C03640=1088.865,407.445,399.289,177.788,26.148,154.195
C03641=1088.871,407.692,399.248,177.791,26.157,154.197
C03642=1088.878,407.938,399.208,177.795,26.166,154.199
C03643=1088.884,408.185,399.168,177.797,26.175,154.200
C03644=1088.890,408.432,399.127,177.800,26.183,154.202
C03645=1088.896,408.678,399.087,177.804,26.192,154.204
C03646=1088.903,408.925,399.047,177.807,26.201,154.206
C03647=1088.909,409.172,399.006,177.811,26.210,154.207
C03648=1088.915,409.419,398.966,177.815,26.219,154.209
C03649=1088.922,409.665,398.925,177.818,26.227,154.211
C03650=1088.927,409.911,398.884,177.821,26.236,154.213
C03651=1088.934,410.158,398.844,177.824,26.245,154.215
C03652=1088.940,410.404,398.804,177.828,26.254,154.217
C03653=1088.946,410.652,398.763,177.831,26.263,154.218
C03654=1088.953,410.879,398.726,177.834,26.272,154.220
C03655=1088.958,411.106,398.688,177.837,26.280,154.222
C03656=1088.963,411.333,398.651,177.841,26.288,154.223
C03657=1088.969,411.560,398.613,177.844,26.297,154.225
C03658=1088.976,411.787,398.575,177.847,26.305,154.227
C03659=1088.981,412.014,398.538,177.850,26.313,154.228
C03660=1088.987,412.241,398.500,177.852,26.322,154.230
C03661=1088.993,412.469,398.463,177.855,26.330,154.232
C03662=1089.000,412.716,398.422,177.859,26.339,154.234
C03663=1089.006,412.962,398.381,177.863,26.349,154.236
C03664=1089.012,413.209,398.340,177.866,26.358,154.238
C03665=1089.019,413.455,398.299,177.869,26.368,154.240
C03666=1089.025,413.702,398.258,177.873,26.377,154.241
C03667=1089.032,413.948,398.218,177.876,26.386,154.243
C03668=1089.038,414.195,398.176,177.880,26.395,154.245
C03669=1089.045,414.441,398.136,177.883,26.405,154.247
C03670=1089.051,414.688,398.094,177.886,26.414,154.249
C03671=1089.058,414.934,398.053,177.890,26.423,154.251
C03672=1089.063,415.181,398.012,177.894,26.433,154.253
C03673=1089.071,415.428,397.971,177.896,26.442,154.255
C03674=1089.077,415.674,397.930,177.900,26.452,154.257
C03675=1089.084,415.921,397.889,177.904,26.462,154.259
C03676=1089.090,416.167,397.848,177.908,26.471,154.261
C03677=1089.096,416.413,397.806,177.910,26.481,154.263
C03678=1089.103,416.660,397.765,177.914,26.490,154.265
C03679=1089.109,416.906,397.723,177.918,26.500,154.267
C03680=1089.115,417.153,397.682,177.921,26.510,154.269
C03681=1089.122,417.399,397.641,177.924,26.520,154.271
C03682=1089.128,417.645,397.599,177.928,26.529,154.273
C03683=1089.135,417.892,397.557,177.931,26.539,154.275
C03684=1089.140,418.138,397.516,177.935,26.549,154.277
C03685=1089.148,418.385,397.475,177.939,26.559,154.279
C03686=1089.154,418.631,397.433,177.941,26.569,154.281
C03687=1089.160,418.878,397.391,177.945,26.579,154.283
C03688=1089.166,419.124,397.350,177.949,26.589,154.285
C03689=1089.173,419.371,397.308,177.952,26.599,154.288
C03690=1089.179,419.617,397.267,177.956,26.609,154.290
C03691=1089.186,419.864,397.226,177.960,26.619,154.292
C03692=1089.192,420.110,397.183,177.963,26.630,154.294
C03693=1089.199,420.356,397.142,177.966,26.639,154.296
C03694=1089.205,420.603,397.100,177.970,26.649,154.298
C03695=1089.211,420.850,397.058,177.973,26.660,154.300
C03696=1089.219,421.096,397.016,177.977,26.670,154.302
C03697=1089.225,421.342,396.975,177.980,26.680,154.305
C03698=1089.231,421.589,396.933,177.984,26.691,154.307
C03699=1089.238,421.834,396.891,177.988,26.701,154.309
C03700=1089.244,422.081,396.849,177.991,26.711,154.311
C03701=1089.251,422.327,396.806,177.995,26.722,154.313
C03702=1089.257,422.574,396.765,177.998,26.732,154.316
C03703=1089.264,422.820,396.722,178.002,26.743,154.318
C03704=1089.270,423.067,396.681,178.006,26.753,154.320
C03705=1089.277,423.312,396.638,178.009,26.764,154.322
C03706=1089.283,423.559,396.597,178.013,26.775,154.324
C03707=1089.290,423.806,396.554,178.016,26.785,154.327
C03708=1089.296,424.051,396.512,178.020,26.796,154.329
C03709=1089.303,424.298,396.470,178.023,26.807,154.331
C03710=1089.311,424.618,396.415,178.027,26.820,154.334
C03711=1089.319,424.939,396.360,178.032,26.834,154.337
C03712=1089.328,425.259,396.305,178.037,26.849,154.340
C03713=1089.336,425.580,396.250,178.042,26.863,154.343
C03714=1089.343,425.825,396.207,178.045,26.874,154.346
C03715=1089.349,426.071,396.165,178.049,26.884,154.348
C03716=1089.356,426.318,396.122,178.052,26.895,154.350
C03717=1089.363,426.564,396.080,178.056,26.906,154.353
C03718=1089.369,426.811,396.037,178.059,26.918,154.355
C03719=1089.376,427.056,395.994,178.063,26.928,154.357
C03720=1089.382,427.302,395.952,178.067,26.940,154.360
C03721=1089.389,427.549,395.909,178.071,26.951,154.362
C03722=1089.396,427.795,395.867,178.074,26.962,154.365
C03723=1089.402,428.042,395.824,178.078,26.973,154.367
C03724=1089.409,428.288,395.781,178.081,26.985,154.369
C03725=1089.415,428.533,395.739,178.085,26.996,154.372
C03726=1089.422,428.780,395.696,178.088,27.007,154.374
C03727=1089.429,429.026,395.653,178.093,27.019,154.377
C03728=1089.436,429.272,395.610,178.096,27.030,154.379
C03729=1089.442,429.518,395.568,178.100,27.041,154.382
C03730=1089.448,429.765,395.524,178.103,27.053,154.384
C03731=1089.456,430.011,395.481,178.107,27.065,154.387
C03732=1089.462,430.257,395.438,178.111,27.076,154.389
C03733=1089.469,430.503,395.395,178.115,27.088,154.392
C03734=1089.474,430.749,395.352,178.118,27.099,154.394
C03735=1089.481,430.995,395.309,178.121,27.111,154.397
C03736=1089.488,431.241,395.266,178.125,27.123,154.399
C03737=1089.495,431.487,395.223,178.129,27.135,154.402
C03738=1089.502,431.733,395.180,178.133,27.146,154.404
C03739=1089.508,431.979,395.137,178.136,27.158,154.407
C03740=1089.515,432.225,395.093,178.141,27.171,154.410
C03741=1089.521,432.472,395.050,178.144,27.182,154.412
C03742=1089.528,432.717,395.007,178.147,27.194,154.415
C03743=1089.535,432.963,394.963,178.151,27.206,154.418
C03744=1089.542,433.210,394.921,178.155,27.218,154.420
C03745=1089.548,433.456,394.877,178.159,27.231,154.423
C03746=1089.554,433.702,394.833,178.162,27.242,154.426
C03747=1089.562,433.947,394.790,178.166,27.255,154.428
C03748=1089.568,434.194,394.747,178.170,27.267,154.431
C03749=1089.575,434.441,394.702,178.173,27.279,154.434
C03750=1089.586,434.835,394.632,178.180,27.300,154.438
C03751=1089.596,435.230,394.562,178.186,27.319,154.442
C03752=1089.607,435.626,394.492,178.192,27.339,154.447
C03753=1089.617,436.021,394.422,178.198,27.359,154.451
C03754=1089.624,436.266,394.378,178.202,27.372,154.454
C03755=1089.631,436.512,394.334,178.205,27.385,154.457
C03756=1089.638,436.759,394.290,178.209,27.398,154.460
C03757=1089.645,437.004,394.246,178.213,27.410,154.463
C03758=1089.651,437.250,394.202,178.217,27.423,154.465
C03759=1089.658,437.496,394.159,178.220,27.436,154.468
C03760=1089.664,437.742,394.114,178.225,27.449,154.471
C03761=1089.671,437.988,394.070,178.228,27.461,154.474
C03762=1089.680,438.310,394.013,178.234,27.479,154.478
C03763=1089.689,438.630,393.955,178.238,27.495,154.481
C03764=1089.698,438.952,393.897,178.244,27.512,154.485
C03765=1089.707,439.273,393.839,178.248,27.529,154.489
C03766=1089.714,439.519,393.796,178.252,27.543,154.492
C03767=1089.720,439.764,393.751,178.256,27.556,154.495
C03768=1089.728,440.010,393.707,178.260,27.569,154.498
C03769=1089.735,440.256,393.663,178.264,27.583,154.501
C03770=1089.742,440.501,393.618,178.268,27.596,154.504
C03771=1089.748,440.748,393.574,178.272,27.609,154.507
C03772=1089.755,440.993,393.529,178.275,27.623,154.510
C03773=1089.762,441.240,393.485,178.279,27.637,154.513
C03774=1089.768,441.485,393.440,178.284,27.650,154.516
C03775=1089.775,441.731,393.396,178.287,27.664,154.519
C03776=1089.782,441.977,393.351,178.291,27.677,154.522
C03777=1089.789,442.222,393.306,178.296,27.691,154.525
C03778=1089.797,442.468,393.261,178.299,27.705,154.529
C03779=1089.803,442.714,393.217,178.303,27.719,154.532
C03780=1089.810,442.959,393.173,178.307,27.733,154.535
C03781=1089.816,443.206,393.127,178.311,27.747,154.538
C03782=1089.823,443.451,393.083,178.315,27.761,154.541
C03783=1089.830,443.697,393.038,178.319,27.775,154.544
C03784=1089.837,443.943,392.993,178.323,27.789,154.547
C03785=1089.844,444.189,392.948,178.327,27.803,154.551
C03786=1089.851,444.434,392.902,178.331,27.817,154.554
C03787=1089.858,444.680,392.857,178.335,27.832,154.557
C03788=1089.865,444.925,392.813,178.338,27.846,154.560
C03789=1089.872,445.171,392.768,178.342,27.860,154.564
C03790=1089.879,445.418,392.722,178.345,27.874,154.567
C03791=1089.886,445.662,392.677,178.348,27.888,154.570
C03792=1089.893,445.908,392.632,178.351,27.903,154.574
C03793=1089.899,446.154,392.587,178.354,27.917,154.577
C03794=1089.907,446.399,392.541,178.356,27.931,154.580
C03795=1089.913,446.646,392.496,178.358,27.945,154.584
C03796=1089.920,446.891,392.451,178.361,27.959,154.587
C03797=1089.928,447.137,392.406,178.363,27.973,154.591
C03798=1089.934,447.383,392.360,178.364,27.987,154.594
C03799=1089.941,447.628,392.315,178.366,28.001,154.597
C03800=1089.948,447.874,392.269,178.367,28.015,154.601
C03801=1089.956,448.119,392.224,178.368,28.030,154.604
C03802=1089.962,448.366,392.178,178.370,28.043,154.608
C03803=1089.969,448.611,392.133,178.371,28.058,154.611
C03804=1089.976,448.857,392.087,178.372,28.071,154.615
C03805=1089.983,449.102,392.042,178.373,28.086,154.618
C03806=1089.990,449.347,391.996,178.373,28.100,154.622
C03807=1089.997,449.593,391.950,178.374,28.114,154.625
C03808=1090.004,449.838,391.906,178.374,28.128,154.629
C03809=1090.015,450.084,391.861,178.374,28.140,154.632
C03810=1089.633,450.077,391.673,178.332,28.336,154.686
C03811=1089.623,449.830,391.716,178.331,28.323,154.682
C03812=1089.615,449.585,391.762,178.330,28.310,154.679
C03813=1089.609,449.340,391.808,178.330,28.295,154.675
C03814=1089.602,449.095,391.853,178.329,28.281,154.672
C03815=1089.594,448.849,391.898,178.329,28.267,154.669
C03816=1089.587,448.603,391.944,178.327,28.253,154.665
C03817=1089.580,448.358,391.990,178.326,28.239,154.662
C03818=1089.573,448.111,392.036,178.325,28.225,154.658
C03819=1089.566,447.867,392.081,178.324,28.211,154.655
C03820=1089.559,447.620,392.126,178.322,28.197,154.651
C03821=1089.552,447.375,392.172,178.320,28.183,154.648
C03822=1089.545,447.128,392.218,178.318,28.169,154.644
C03823=1089.538,446.884,392.263,178.316,28.154,154.641
C03824=1089.532,446.637,392.308,178.314,28.140,154.637
C03825=1089.524,446.392,392.354,178.311,28.126,154.634
C03826=1089.517,446.146,392.399,178.309,28.111,154.631
C03827=1089.510,445.901,392.445,178.306,28.097,154.627
C03828=1089.503,445.655,392.490,178.303,28.083,154.624
C03829=1089.497,445.409,392.535,178.300,28.069,154.621
C03830=1089.489,445.164,392.581,178.296,28.055,154.617
C03831=1089.482,444.918,392.626,178.293,28.040,154.614
C03832=1089.475,444.672,392.670,178.289,28.027,154.611
C03833=1089.468,444.426,392.716,178.285,28.012,154.607
C03834=1089.462,444.181,392.761,178.281,27.998,154.604
C03835=1089.454,443.935,392.806,178.277,27.984,154.601
C03836=1089.448,443.690,392.850,178.273,27.969,154.598
C03837=1089.441,443.443,392.896,178.269,27.955,154.595
C03838=1089.434,443.198,392.940,178.264,27.941,154.591
C03839=1089.427,442.952,392.985,178.261,27.927,154.588
C03840=1089.420,442.707,393.030,178.257,27.913,154.585
C03841=1089.413,442.460,393.075,178.252,27.899,154.582
C03842=1089.406,442.215,393.119,178.249,27.886,154.579
C03843=1089.400,441.969,393.165,178.245,27.872,154.576
C03844=1089.393,441.723,393.210,178.240,27.858,154.573
C03845=1089.385,441.477,393.255,178.237,27.844,154.570
C03846=1089.379,441.232,393.299,178.233,27.831,154.567
C03847=1089.372,440.986,393.343,178.229,27.817,154.563
C03848=1089.365,440.740,393.388,178.225,27.803,154.560
C03849=1089.358,440.495,393.432,178.220,27.790,154.557
C03850=1089.351,440.249,393.477,178.217,27.777,154.554
C03851=1089.345,440.003,393.521,178.213,27.763,154.551
C03852=1089.338,439.757,393.566,178.209,27.750,154.548
C03853=1089.331,439.511,393.610,178.205,27.736,154.545
C03854=1089.324,439.265,393.655,178.201,27.723,154.542
C03855=1089.315,438.957,393.710,178.196,27.707,154.539
C03856=1089.307,438.648,393.765,178.191,27.690,154.535
C03857=1089.298,438.340,393.821,178.186,27.674,154.531
C03858=1089.290,438.031,393.876,178.181,27.658,154.528
C03859=1089.283,437.785,393.920,178.177,27.645,154.525
C03860=1089.275,437.540,393.964,178.174,27.632,154.522
C03861=1089.269,437.294,394.008,178.169,27.619,154.519
C03862=1089.262,437.048,394.052,178.166,27.606,154.516
C03863=1089.255,436.801,394.096,178.162,27.593,154.514
C03864=1089.249,436.556,394.141,178.158,27.581,154.511
C03865=1089.241,436.310,394.184,178.154,27.568,154.508
C03866=1089.235,436.064,394.228,178.150,27.555,154.505
C03867=1089.229,435.818,394.272,178.146,27.543,154.502
C03868=1089.222,435.572,394.316,178.142,27.530,154.500
C03869=1089.214,435.326,394.359,178.139,27.518,154.497
C03870=1089.208,435.080,394.403,178.135,27.505,154.494
C03871=1089.202,434.834,394.447,178.131,27.493,154.491
C03872=1089.195,434.588,394.491,178.127,27.480,154.489
C03873=1089.188,434.342,394.534,178.124,27.468,154.486
C03874=1089.181,434.096,394.578,178.119,27.456,154.483
C03875=1089.175,433.850,394.622,178.116,27.443,154.480
C03876=1089.168,433.605,394.665,178.112,27.431,154.478
C03877=1089.161,433.359,394.709,178.108,27.419,154.475
C03878=1089.155,433.112,394.752,178.104,27.407,154.472
C03879=1089.149,432.866,394.796,178.101,27.394,154.470
C03880=1089.141,432.620,394.840,178.096,27.382,154.467
C03881=1089.135,432.373,394.883,178.093,27.371,154.464
C03882=1089.128,432.127,394.926,178.089,27.358,154.462
C03883=1089.121,431.882,394.970,178.085,27.346,154.459
C03884=1089.115,431.635,395.012,178.081,27.335,154.457
C03885=1089.108,431.389,395.056,178.078,27.323,154.454
C03886=1089.101,431.143,395.099,178.074,27.311,154.451
C03887=1089.094,430.897,395.142,178.071,27.299,154.449
C03888=1089.088,430.651,395.185,178.066,27.287,154.446
C03889=1089.081,430.405,395.228,178.063,27.276,154.444
C03890=1089.075,430.158,395.271,178.059,27.264,154.441
C03891=1089.068,429.913,395.315,178.056,27.253,154.439
C03892=1089.062,429.667,395.357,178.051,27.241,154.436
C03893=1089.055,429.421,395.400,178.048,27.230,154.434
C03894=1089.048,429.175,395.443,178.044,27.218,154.431
C03895=1089.042,428.928,395.486,178.041,27.206,154.429
C03896=1089.035,428.682,395.529,178.037,27.195,154.426
C03897=1089.028,428.436,395.572,178.033,27.184,154.424
C03898=1089.022,428.190,395.615,178.030,27.172,154.421
C03899=1089.015,427.944,395.658,178.025,27.161,154.419
C03900=1089.008,427.697,395.700,178.022,27.150,154.417
C03901=1089.001,427.451,395.743,178.018,27.139,154.414
C03902=1088.996,427.205,395.786,178.015,27.128,154.412
C03903=1088.989,426.959,395.828,178.011,27.116,154.409
C03904=1088.982,426.713,395.871,178.007,27.106,154.407
C03905=1088.975,426.466,395.913,178.004,27.094,154.405
C03906=1088.968,426.220,395.956,178.000,27.083,154.402
C03907=1088.962,425.984,395.996,177.996,27.073,154.400
C03908=1088.956,425.750,396.037,177.993,27.062,154.398
C03909=1088.950,425.514,396.078,177.989,27.052,154.396
C03910=1088.944,425.279,396.118,177.986,27.042,154.393
C03911=1088.937,425.044,396.159,177.983,27.031,154.391
C03912=1088.931,424.809,396.199,177.979,27.021,154.389
C03913=1088.925,424.572,396.240,177.975,27.010,154.387
C03914=1088.919,424.337,396.281,177.972,27.000,154.384
C03915=1088.912,424.091,396.323,177.969,26.989,154.382
C03916=1088.906,423.845,396.365,177.965,26.979,154.380
C03917=1088.899,423.598,396.407,177.962,26.968,154.378
C03918=1088.893,423.353,396.449,177.958,26.958,154.375
C03919=1088.886,423.106,396.492,177.954,26.947,154.373
C03920=1088.879,422.859,396.534,177.951,26.936,154.371
C03921=1088.873,422.614,396.576,177.947,26.925,154.369
C03922=1088.867,422.367,396.618,177.943,26.915,154.366
C03923=1088.860,422.121,396.660,177.940,26.904,154.364
C03924=1088.854,421.874,396.702,177.936,26.894,154.362
C03925=1088.847,421.628,396.744,177.932,26.884,154.360
C03926=1088.840,421.381,396.786,177.929,26.873,154.358
C03927=1088.834,421.136,396.828,177.925,26.863,154.355
C03928=1088.828,420.889,396.870,177.921,26.853,154.353
C03929=1088.821,420.643,396.911,177.918,26.843,154.351
C03930=1088.814,420.397,396.953,177.915,26.832,154.349
C03931=1088.807,420.150,396.995,177.911,26.822,154.347
C03932=1088.802,419.903,397.037,177.907,26.812,154.345
C03933=1088.795,419.657,397.079,177.904,26.802,154.343
C03934=1088.789,419.411,397.121,177.900,26.792,154.341
C03935=1088.781,419.164,397.162,177.896,26.781,154.338
C03936=1088.775,418.918,397.203,177.894,26.772,154.336
C03937=1088.769,418.671,397.245,177.890,26.762,154.334
C03938=1088.763,418.425,397.287,177.886,26.752,154.332
C03939=1088.756,418.178,397.328,177.882,26.742,154.330
C03940=1088.750,417.932,397.369,177.879,26.732,154.328
C03941=1088.743,417.685,397.411,177.876,26.722,154.326
C03942=1088.737,417.439,397.453,177.872,26.712,154.324
C03943=1088.730,417.181,397.497,177.869,26.702,154.322
C03944=1088.723,416.924,397.539,177.865,26.691,154.320
C03945=1088.717,416.666,397.583,177.861,26.681,154.317
C03946=1088.710,416.408,397.627,177.858,26.671,154.315
C03947=1088.704,416.162,397.668,177.854,26.661,154.313
C03948=1088.698,415.915,397.708,177.850,26.652,154.311
C03949=1088.691,415.669,397.750,177.847,26.643,154.309
C03950=1088.684,415.423,397.791,177.844,26.633,154.307
C03951=1088.678,415.176,397.833,177.840,26.623,154.305
C03952=1088.671,414.930,397.874,177.837,26.614,154.303
C03953=1088.665,414.682,397.915,177.833,26.604,154.301
C03954=1088.658,414.436,397.956,177.829,26.595,154.300
C03955=1088.652,414.190,397.998,177.826,26.585,154.298
C03956=1088.645,413.943,398.038,177.823,26.576,154.296
C03957=1088.639,413.697,398.079,177.819,26.567,154.294
C03958=1088.632,413.450,398.120,177.816,26.557,154.292
C03959=1088.626,413.204,398.161,177.812,26.548,154.290
C03960=1088.620,412.957,398.202,177.809,26.539,154.288
C03961=1088.613,412.710,398.243,177.806,26.530,154.286
C03962=1088.607,412.464,398.284,177.802,26.520,154.284
C03963=1088.602,412.241,398.320,177.799,26.512,154.283
C03964=1088.595,412.020,398.357,177.796,26.504,154.281
C03965=1088.589,411.798,398.394,177.793,26.495,154.279
C03966=1088.584,411.575,398.430,177.790,26.487,154.278
C03967=1088.578,411.353,398.467,177.787,26.479,154.276
C03968=1088.572,411.131,398.504,177.784,26.471,154.274
C03969=1088.567,410.909,398.540,177.780,26.463,154.273
C03970=1088.561,410.687,398.578,177.777,26.455,154.271
C03971=1088.555,410.440,398.618,177.774,26.445,154.269
C03972=1088.548,410.194,398.659,177.771,26.437,154.267
C03973=1088.542,409.948,398.699,177.767,26.427,154.265
C03974=1088.535,409.700,398.740,177.764,26.419,154.264
C03975=1088.529,409.454,398.780,177.760,26.410,154.262
C03976=1088.523,409.207,398.821,177.757,26.401,154.260
C03977=1088.517,408.961,398.862,177.753,26.392,154.258
C03978=1088.510,408.715,398.902,177.750,26.383,154.256
C03979=1088.505,408.468,398.943,177.747,26.374,154.255
C03980=1088.498,408.221,398.983,177.744,26.365,154.253
C03981=1088.492,407.975,399.023,177.740,26.357,154.251
C03982=1088.486,407.727,399.064,177.737,26.348,154.249
C03983=1088.479,407.481,399.104,177.733,26.339,154.247
C03984=1088.473,407.234,399.144,177.730,26.331,154.246
C03985=1088.467,406.988,399.184,177.726,26.321,154.244
C03986=1088.460,406.741,399.225,177.723,26.313,154.242
C03987=1088.455,406.494,399.265,177.720,26.305,154.241
C03988=1088.448,406.248,399.305,177.716,26.296,154.239
C03989=1088.442,406.001,399.346,177.713,26.288,154.237
C03990=1088.435,405.755,399.386,177.710,26.278,154.235
C03991=1088.429,405.508,399.425,177.707,26.271,154.234
C03992=1088.423,405.261,399.465,177.704,26.262,154.232
C03993=1088.416,405.014,399.506,177.700,26.254,154.230
C03994=1088.410,404.767,399.546,177.697,26.245,154.229
C03995=1088.403,404.520,399.585,177.693,26.236,154.227
C03996=1088.397,404.274,399.626,177.690,26.228,154.225
C03997=1088.391,404.027,399.666,177.687,26.220,154.224
C03998=1088.384,403.781,399.706,177.683,26.211,154.222
C03999=1088.378,403.534,399.745,177.680,26.203,154.220
C04000=1088.372,403.287,399.785,177.677,26.195,154.219
C04001=1088.366,403.040,399.825,177.673,26.187,154.217
C04002=1088.359,402.794,399.865,177.670,26.178,154.215
C04003=1088.353,402.547,399.905,177.667,26.171,154.214
C04004=1088.347,402.300,399.945,177.663,26.162,154.212
C04005=1088.341,402.054,399.984,177.660,26.154,154.211
C04006=1088.335,401.807,400.024,177.657,26.146,154.209
C04007=1088.329,401.560,400.064,177.653,26.138,154.207
C04008=1088.322,401.314,400.103,177.650,26.130,154.206
C04009=1088.316,401.066,400.142,177.647,26.122,154.204
C04010=1088.309,400.820,400.182,177.644,26.114,154.203
C04011=1088.303,400.573,400.222,177.640,26.106,154.201
C04012=1088.297,400.326,400.262,177.637,26.098,154.200
C04013=1088.291,400.079,400.301,177.634,26.090,154.198
C04014=1088.285,399.833,400.340,177.631,26.082,154.196
C04015=1088.278,399.587,400.380,177.627,26.074,154.195
C04016=1088.272,399.339,400.419,177.624,26.066,154.193
C04017=1088.266,399.092,400.459,177.621,26.058,154.192
C04018=1088.260,398.845,400.498,177.618,26.050,154.190
C04019=1088.255,398.618,400.534,177.615,26.043,154.189
C04020=1088.249,398.392,400.571,177.611,26.036,154.187
C04021=1088.243,398.164,400.607,177.608,26.029,154.186
C04022=1088.237,397.938,400.643,177.606,26.022,154.185
C04023=1088.231,397.711,400.679,177.603,26.015,154.183
C04024=1088.225,397.483,400.715,177.600,26.007,154.182
C04025=1088.220,397.256,400.751,177.596,26.000,154.181
C04026=1088.214,397.029,400.787,177.593,25.993,154.179
C04027=1088.208,396.782,400.826,177.590,25.985,154.178
C04028=1088.202,396.535,400.866,177.587,25.978,154.176
C04029=1088.195,396.288,400.904,177.584,25.970,154.175
C04030=1088.190,396.041,400.944,177.581,25.963,154.173
C04031=1088.183,395.795,400.982,177.578,25.955,154.172
C04032=1088.177,395.547,401.022,177.574,25.947,154.170
C04033=1088.171,395.301,401.061,177.570,25.940,154.169
C04034=1088.164,395.054,401.100,177.567,25.932,154.167
C04035=1088.158,394.807,401.139,177.564,25.925,154.166
C04036=1088.152,394.561,401.178,177.561,25.917,154.165
C04037=1088.146,394.314,401.217,177.558,25.910,154.163
C04038=1088.139,394.067,401.256,177.555,25.902,154.162
C04039=1088.134,393.820,401.294,177.552,25.895,154.160
C04040=1088.127,393.573,401.333,177.548,25.888,154.159
C04041=1088.121,393.326,401.372,177.545,25.880,154.157
C04042=1088.115,393.080,401.411,177.541,25.873,154.156
C04043=1088.109,392.832,401.449,177.538,25.866,154.155
C04044=1088.103,392.586,401.488,177.535,25.858,154.153
C04045=1088.096,392.339,401.527,177.532,25.851,154.152
C04046=1088.091,392.092,401.565,177.529,25.844,154.150
C04047=1088.084,391.845,401.604,177.526,25.836,154.149
C04048=1088.077,391.598,401.643,177.522,25.829,154.148
C04049=1088.072,391.352,401.681,177.519,25.822,154.146
C04050=1088.065,391.105,401.720,177.516,25.815,154.145
C04051=1088.060,390.858,401.758,177.512,25.807,154.144
C04052=1088.053,390.611,401.797,177.509,25.800,154.142
C04053=1088.046,390.364,401.836,177.506,25.793,154.141
C04054=1088.041,390.117,401.874,177.502,25.786,154.140
C04055=1088.034,389.870,401.913,177.499,25.779,154.138
C04056=1088.028,389.624,401.951,177.496,25.772,154.137
C04057=1088.022,389.376,401.989,177.493,25.765,154.136
C04058=1088.015,389.130,402.027,177.490,25.758,154.134
C04059=1088.009,388.883,402.065,177.486,25.751,154.133
C04060=1088.003,388.636,402.104,177.483,25.744,154.132
C04061=1087.997,388.389,402.142,177.480,25.737,154.131
C04062=1087.991,388.142,402.180,177.477,25.730,154.129
C04063=1087.985,387.896,402.219,177.474,25.723,154.128
C04064=1087.978,387.648,402.257,177.470,25.716,154.127
C04065=1087.972,387.402,402.295,177.467,25.709,154.125
C04066=1087.966,387.155,402.333,177.464,25.703,154.124
C04067=1087.960,386.908,402.372,177.461,25.696,154.123
C04068=1087.954,386.661,402.410,177.458,25.689,154.122
C04069=1087.948,386.414,402.448,177.454,25.682,154.120
C04070=1087.942,386.167,402.485,177.451,25.675,154.119
C04071=1087.936,385.921,402.524,177.448,25.668,154.118
C04072=1087.929,385.673,402.562,177.445,25.661,154.116
C04073=1087.923,385.427,402.600,177.441,25.655,154.115
C04074=1087.918,385.180,402.638,177.438,25.648,154.114
C04075=1087.912,384.959,402.672,177.435,25.641,154.113
C04076=1087.907,384.738,402.706,177.432,25.636,154.112
C04077=1087.901,384.519,402.739,177.430,25.630,154.111
C04078=1087.896,384.297,402.773,177.426,25.623,154.110
C04079=1087.891,384.077,402.807,177.424,25.618,154.108
C04080=1087.886,383.857,402.841,177.421,25.611,154.107
C04081=1087.879,383.637,402.874,177.418,25.606,154.106
C04082=1087.874,383.417,402.909,177.416,25.600,154.105
C04083=1087.868,383.170,402.946,177.412,25.593,154.104
C04084=1087.862,382.922,402.984,177.409,25.586,154.103
C04085=1087.856,382.675,403.022,177.406,25.580,154.102
C04086=1087.850,382.429,403.059,177.403,25.573,154.100
C04087=1087.844,382.181,403.097,177.399,25.566,154.099
C04088=1087.838,381.934,403.135,177.396,25.560,154.098
C04089=1087.831,381.688,403.172,177.393,25.554,154.097
C04090=1087.826,381.441,403.210,177.389,25.547,154.096
C04091=1087.819,381.193,403.247,177.386,25.540,154.095
C04092=1087.813,380.946,403.285,177.383,25.534,154.093
C04093=1087.807,380.700,403.322,177.380,25.528,154.092
C04094=1087.801,380.453,403.359,177.377,25.521,154.091
C04095=1087.795,380.205,403.398,177.374,25.515,154.090
C04096=1087.789,379.958,403.435,177.370,25.509,154.089
C04097=1087.783,379.711,403.472,177.367,25.502,154.088
C04098=1087.777,379.465,403.510,177.364,25.496,154.087
C04099=1087.771,379.218,403.547,177.360,25.489,154.085
C04100=1087.764,378.970,403.585,177.357,25.483,154.084
C04101=1087.758,378.723,403.622,177.355,25.477,154.083
C04102=1087.752,378.476,403.659,177.351,25.471,154.082
C04103=1087.746,378.229,403.697,177.348,25.464,154.081
C04104=1087.741,377.982,403.734,177.345,25.458,154.080
C04105=1087.734,377.735,403.771,177.342,25.451,154.079
C04106=1087.728,377.487,403.808,177.338,25.445,154.077
C04107=1087.722,377.241,403.846,177.335,25.439,154.076
C04108=1087.716,376.994,403.882,177.332,25.433,154.075
C04109=1087.710,376.747,403.920,177.329,25.427,154.074
C04110=1087.704,376.500,403.957,177.326,25.420,154.073
C04111=1087.698,376.252,403.994,177.322,25.414,154.072
C04112=1087.692,376.006,404.031,177.319,25.408,154.071
C04113=1087.686,375.758,404.068,177.317,25.402,154.070
C04114=1087.680,375.511,404.105,177.313,25.396,154.069
C04115=1087.674,375.265,404.143,177.310,25.389,154.068
C04116=1087.668,375.017,404.180,177.306,25.383,154.067
C04117=1087.662,374.770,404.216,177.303,25.377,154.066
C04118=1087.656,374.523,404.253,177.301,25.371,154.064
C04119=1087.651,374.276,404.291,177.297,25.365,154.063
C04120=1087.644,374.029,404.327,177.294,25.358,154.062
C04121=1087.638,373.781,404.365,177.291,25.353,154.061
C04122=1087.632,373.534,404.401,177.287,25.347,154.060
C04123=1087.625,373.287,404.438,177.285,25.341,154.059
C04124=1087.620,373.039,404.475,177.281,25.335,154.058
C04125=1087.613,372.792,404.511,177.278,25.329,154.057
C04126=1087.608,372.546,404.549,177.275,25.323,154.056
C04127=1087.601,372.299,404.585,177.272,25.317,154.055
C04128=1087.595,372.052,404.622,177.269,25.311,154.054
C04129=1087.589,371.804,404.659,177.265,25.305,154.053
C04130=1087.583,371.557,404.695,177.262,25.299,154.052
C04131=1087.573,371.144,404.756,177.257,25.289,154.050
C04132=1087.563,370.731,404.818,177.251,25.279,154.049
C04133=1087.553,370.318,404.879,177.247,25.270,154.047
C04134=1087.543,369.906,404.940,177.241,25.260,154.045
C04135=1087.536,369.659,404.976,177.238,25.254,154.044
C04136=1087.531,369.411,405.012,177.234,25.248,154.043
C04137=1087.525,369.164,405.049,177.231,25.242,154.042
C04138=1087.518,368.917,405.085,177.229,25.237,154.041
C04139=1087.513,368.669,405.122,177.225,25.231,154.040
C04140=1087.507,368.422,405.158,177.222,25.225,154.039
C04141=1087.501,368.175,405.194,177.219,25.220,154.038
C04142=1087.495,367.928,405.231,177.216,25.214,154.037
C04143=1087.489,367.681,405.268,177.212,25.208,154.036
C04144=1087.483,367.433,405.303,177.210,25.202,154.035
C04145=1087.477,367.186,405.340,177.206,25.197,154.034
C04146=1087.471,366.939,405.377,177.203,25.191,154.034
C04147=1087.466,366.692,405.412,177.200,25.186,154.033
C04148=1087.459,366.445,405.449,177.197,25.179,154.032
C04149=1087.453,366.197,405.484,177.194,25.174,154.031
C04150=1087.448,365.950,405.521,177.191,25.168,154.030
C04151=1087.442,365.702,405.557,177.188,25.163,154.029
C04152=1087.436,365.456,405.593,177.184,25.157,154.028
C04153=1087.430,365.208,405.629,177.182,25.151,154.027
C04154=1087.424,364.961,405.665,177.178,25.146,154.026
C04155=1087.418,364.713,405.701,177.175,25.140,154.025
C04156=1087.411,364.466,405.738,177.172,25.135,154.024
C04157=1087.405,364.219,405.773,177.169,25.129,154.023
C04158=1087.400,363.972,405.810,177.165,25.124,154.022
C04159=1087.394,363.724,405.846,177.163,25.118,154.021
C04160=1087.388,363.477,405.881,177.159,25.113,154.020
C04161=1087.382,363.229,405.918,177.156,25.107,154.020
C04162=1087.376,362.982,405.954,177.153,25.102,154.019
C04163=1087.370,362.735,405.989,177.150,25.096,154.018
C04164=1087.364,362.488,406.025,177.146,25.091,154.017
C04165=1087.358,362.240,406.061,177.143,25.086,154.016
C04166=1087.352,361.992,406.097,177.140,25.080,154.015
C04167=1087.347,361.745,406.132,177.137,25.075,154.014
C04168=1087.339,361.499,406.168,177.134,25.069,154.013
C04169=1087.333,361.251,406.204,177.130,25.064,154.013
C04170=1087.327,361.003,406.240,177.128,25.059,154.012
C04171=1087.322,360.756,406.275,177.124,25.053,154.011
C04172=1087.316,360.509,406.311,177.122,25.048,154.010
C04173=1087.310,360.262,406.347,177.118,25.042,154.009
C04174=1087.304,360.015,406.382,177.115,25.037,154.008
C04175=1087.298,359.767,406.418,177.112,25.032,154.007
C04176=1087.292,359.519,406.454,177.109,25.026,154.006
C04177=1087.287,359.272,406.489,177.106,25.021,154.006
C04178=1087.280,359.025,406.524,177.102,25.016,154.005
C04179=1087.274,358.777,406.560,177.099,25.010,154.004
C04180=1087.268,358.530,406.596,177.096,25.005,154.003
C04181=1087.262,358.283,406.631,177.093,25.000,154.002
C04182=1087.256,358.035,406.667,177.090,24.995,154.001
C04183=1087.247,357.638,406.723,177.084,24.986,154.000
C04184=1087.237,357.241,406.780,177.080,24.978,153.999
C04185=1087.227,356.843,406.837,177.075,24.970,153.997
C04186=1087.218,356.446,406.894,177.069,24.961,153.996
C04187=1087.212,356.199,406.929,177.067,24.956,153.995
C04188=1087.206,355.952,406.965,177.063,24.951,153.994
C04189=1087.200,355.705,406.999,177.061,24.946,153.993
C04190=1087.195,355.457,407.034,177.057,24.941,153.993
C04191=1087.189,355.209,407.070,177.054,24.936,153.992
C04192=1087.182,354.962,407.105,177.051,24.930,153.991
C04193=1087.176,354.715,407.141,177.048,24.926,153.990
C04194=1087.171,354.467,407.175,177.045,24.920,153.989
C04195=1087.164,354.220,407.210,177.042,24.915,153.989
C04196=1087.159,353.973,407.246,177.038,24.910,153.988
C04197=1087.153,353.724,407.281,177.036,24.905,153.987
C04198=1087.147,353.478,407.316,177.032,24.900,153.986
C04199=1087.141,353.230,407.351,177.030,24.895,153.985
C04200=1087.136,352.982,407.386,177.026,24.890,153.985
C04201=1087.129,352.735,407.421,177.023,24.885,153.984
C04202=1087.124,352.487,407.456,177.020,24.880,153.983
C04203=1087.117,352.240,407.491,177.017,24.875,153.982
C04204=1087.112,351.992,407.526,177.013,24.870,153.982
C04205=1087.105,351.745,407.561,177.011,24.865,153.981
C04206=1087.100,351.498,407.595,177.007,24.860,153.980
C04207=1087.094,351.250,407.630,177.005,24.855,153.979
C04208=1087.088,351.003,407.665,177.001,24.850,153.979
C04209=1087.082,350.755,407.700,176.998,24.845,153.978
C04210=1087.077,350.508,407.735,176.995,24.840,153.977
C04211=1087.070,350.260,407.769,176.992,24.836,153.976
C04212=1087.065,350.013,407.805,176.988,24.830,153.975
C04213=1087.058,349.765,407.839,176.986,24.826,153.975
C04214=1087.053,349.518,407.874,176.982,24.820,153.974
C04215=1087.046,349.270,407.909,176.979,24.816,153.973
C04216=1087.040,349.022,407.943,176.976,24.811,153.972
C04217=1087.035,348.775,407.978,176.973,24.806,153.972
C04218=1087.029,348.527,408.013,176.970,24.801,153.971
C04219=1087.023,348.280,408.047,176.967,24.796,153.970
C04220=1087.017,348.032,408.082,176.964,24.792,153.969
C04221=1087.011,347.785,408.116,176.961,24.786,153.969
C04222=1087.006,347.538,408.151,176.958,24.782,153.968
C04223=1086.999,347.290,408.186,176.954,24.777,153.967
C04224=1086.993,347.042,408.220,176.951,24.772,153.967
C04225=1086.988,346.794,408.255,176.948,24.767,153.966
C04226=1086.982,346.547,408.289,176.945,24.762,153.965
C04227=1086.976,346.300,408.323,176.942,24.758,153.964
C04228=1086.970,346.051,408.358,176.939,24.753,153.964
C04229=1086.964,345.805,408.393,176.936,24.748,153.963
C04230=1086.958,345.557,408.427,176.932,24.743,153.962
C04231=1086.952,345.309,408.462,176.930,24.739,153.962
C04232=1086.947,345.062,408.496,176.927,24.734,153.961
C04233=1086.941,344.814,408.530,176.923,24.729,153.960
C04234=1086.934,344.566,408.564,176.921,24.724,153.959
C04235=1086.925,344.172,408.618,176.916,24.717,153.958
C04236=1086.916,343.778,408.673,176.911,24.710,153.957
C04237=1086.906,343.383,408.728,176.906,24.702,153.956
C04238=1086.897,342.989,408.782,176.901,24.695,153.955
C04239=1086.891,342.741,408.816,176.897,24.690,153.954
C04240=1086.885,342.494,408.850,176.895,24.685,153.954
C04241=1086.880,342.246,408.885,176.892,24.681,153.953
C04242=1086.874,341.999,408.919,176.888,24.676,153.952
C04243=1086.868,341.751,408.952,176.885,24.672,153.952
C04244=1086.862,341.503,408.987,176.883,24.667,153.951
C04245=1086.856,341.255,409.021,176.879,24.662,153.950
C04246=1086.850,341.008,409.055,176.876,24.658,153.950
C04247=1086.844,340.760,409.088,176.873,24.653,153.949
C04248=1086.839,340.513,409.122,176.870,24.648,153.948
C04249=1086.832,340.265,409.156,176.867,24.644,153.948
C04250=1086.827,340.017,409.190,176.863,24.640,153.947
C04251=1086.821,339.770,409.224,176.861,24.635,153.946
C04252=1086.815,339.522,409.258,176.858,24.631,153.946
C04253=1086.809,339.275,409.291,176.854,24.626,153.945
C04254=1086.803,339.027,409.326,176.851,24.621,153.944
C04255=1086.797,338.779,409.360,176.849,24.617,153.944
C04256=1086.791,338.531,409.393,176.845,24.612,153.943
C04257=1086.786,338.284,409.427,176.842,24.608,153.942
C04258=1086.780,338.036,409.460,176.839,24.604,153.942
C04259=1086.774,337.789,409.495,176.836,24.599,153.941
C04260=1086.768,337.540,409.528,176.833,24.594,153.940
C04261=1086.762,337.293,409.562,176.830,24.590,153.940
C04262=1086.757,337.045,409.596,176.827,24.585,153.939
C04263=1086.751,336.798,409.630,176.824,24.581,153.938
C04264=1086.745,336.550,409.663,176.821,24.577,153.938
C04265=1086.739,336.303,409.696,176.818,24.572,153.937
C04266=1086.733,336.055,409.730,176.814,24.568,153.937
C04267=1086.727,335.807,409.763,176.812,24.564,153.936
C04268=1086.721,335.559,409.798,176.809,24.559,153.935
C04269=1086.715,335.311,409.831,176.805,24.555,153.935
C04270=1086.709,335.064,409.864,176.802,24.550,153.934
C04271=1086.703,334.816,409.898,176.799,24.546,153.933
C04272=1086.698,334.568,409.931,176.796,24.541,153.933
C04273=1086.692,334.321,409.964,176.793,24.537,153.932
C04274=1086.686,334.073,409.998,176.790,24.533,153.932
C04275=1086.680,333.826,410.031,176.788,24.528,153.931
C04276=1086.674,333.578,410.064,176.784,24.524,153.930
C04277=1086.669,333.330,410.098,176.781,24.519,153.930
C04278=1086.663,333.083,410.132,176.778,24.515,153.929
C04279=1086.657,332.835,410.165,176.775,24.511,153.928
C04280=1086.651,332.587,410.198,176.772,24.507,153.928
C04281=1086.646,332.339,410.231,176.769,24.502,153.927
C04282=1086.640,332.091,410.265,176.766,24.498,153.927
C04283=1086.634,331.844,410.297,176.763,24.494,153.926
C04284=1086.628,331.596,410.331,176.760,24.489,153.925
C04285=1086.622,331.348,410.365,176.757,24.485,153.925
C04286=1086.616,331.101,410.398,176.754,24.481,153.924
C04287=1086.606,330.700,410.451,176.749,24.475,153.923
C04288=1086.596,330.300,410.504,176.744,24.467,153.922
C04289=1086.587,329.900,410.558,176.739,24.461,153.922
C04290=1086.577,329.500,410.611,176.733,24.454,153.921
C04291=1086.571,329.252,410.644,176.731,24.450,153.920
C04292=1086.566,329.004,410.677,176.728,24.446,153.920
C04293=1086.559,328.757,410.710,176.725,24.442,153.919
C04294=1086.554,328.509,410.743,176.722,24.438,153.918
C04295=1086.547,328.261,410.776,176.718,24.433,153.918
C04296=1086.541,328.013,410.808,176.715,24.429,153.917
C04297=1086.536,327.765,410.841,176.713,24.425,153.917
C04298=1086.530,327.518,410.874,176.710,24.421,153.916
C04299=1086.524,327.270,410.907,176.706,24.417,153.916
C04300=1086.518,327.022,410.940,176.703,24.412,153.915
C04301=1086.511,326.774,410.973,176.700,24.408,153.914
C04302=1086.507,326.527,411.005,176.698,24.404,153.914
C04303=1086.501,326.279,411.038,176.695,24.400,153.913
C04304=1086.495,326.031,411.071,176.692,24.396,153.913
C04305=1086.489,325.784,411.104,176.688,24.392,153.912
C04306=1086.483,325.535,411.136,176.685,24.388,153.912
C04307=1086.477,325.287,411.169,176.682,24.384,153.911
C04308=1086.471,325.040,411.202,176.679,24.380,153.911
C04309=1086.465,324.792,411.234,176.677,24.376,153.910
C04310=1086.460,324.544,411.267,176.673,24.371,153.910
C04311=1086.454,324.297,411.300,176.670,24.367,153.909
C04312=1086.448,324.049,411.332,176.667,24.363,153.908
C04313=1086.442,323.801,411.365,176.664,24.359,153.908
C04314=1086.436,323.552,411.397,176.661,24.355,153.907
C04315=1086.430,323.305,411.430,176.659,24.351,153.907
C04316=1086.425,323.058,411.463,176.655,24.347,153.906
C04317=1086.419,322.809,411.495,176.652,24.343,153.906
C04318=1086.413,322.562,411.528,176.649,24.339,153.905
C04319=1086.407,322.313,411.560,176.646,24.335,153.905
C04320=1086.402,322.066,411.593,176.643,24.331,153.904
C04321=1086.396,321.818,411.625,176.640,24.327,153.904
C04322=1086.389,321.571,411.657,176.638,24.323,153.903
C04323=1086.384,321.322,411.690,176.634,24.319,153.903
C04324=1086.379,321.075,411.722,176.631,24.314,153.902
C04325=1086.372,320.827,411.754,176.628,24.310,153.901
C04326=1086.367,320.578,411.787,176.625,24.306,153.901
C04327=1086.361,320.332,411.819,176.622,24.303,153.901
C04328=1086.355,320.083,411.852,176.619,24.299,153.900
C04329=1086.349,319.835,411.884,176.617,24.295,153.899
C04330=1086.343,319.588,411.916,176.614,24.291,153.899
C04331=1086.339,319.340,411.949,176.610,24.286,153.898
C04332=1086.333,319.092,411.981,176.607,24.282,153.898
C04333=1086.327,318.845,412.013,176.604,24.279,153.897
C04334=1086.321,318.596,412.045,176.601,24.275,153.897
C04335=1086.316,318.348,412.078,176.598,24.271,153.896
C04336=1086.310,318.100,412.109,176.596,24.267,153.896
C04337=1086.304,317.853,412.142,176.593,24.263,153.895
C04338=1086.298,317.605,412.174,176.590,24.259,153.895
C04339=1086.289,317.198,412.226,176.585,24.252,153.894
C04340=1086.280,316.790,412.279,176.580,24.246,153.893
C04341=1086.270,316.384,412.332,176.574,24.239,153.892
C04342=1086.261,315.977,412.385,176.570,24.233,153.891
C04343=1086.256,315.729,412.417,176.567,24.229,153.891
C04344=1086.250,315.481,412.449,176.564,24.225,153.890
C04345=1086.244,315.234,412.480,176.561,24.221,153.890
C04346=1086.238,314.986,412.512,176.558,24.217,153.889
C04347=1086.233,314.738,412.544,176.555,24.213,153.889
C04348=1086.227,314.490,412.576,176.552,24.209,153.888
C04349=1086.221,314.242,412.608,176.549,24.205,153.888
C04350=1086.215,313.994,412.640,176.546,24.202,153.887
C04351=1086.209,313.746,412.671,176.543,24.198,153.887
C04352=1086.203,313.498,412.703,176.540,24.194,153.886
C04353=1086.197,313.250,412.735,176.537,24.190,153.886
C04354=1086.191,313.002,412.767,176.534,24.187,153.886
C04355=1086.185,312.755,412.798,176.531,24.183,153.885
C04356=1086.179,312.507,412.830,176.529,24.179,153.885
C04357=1086.174,312.258,412.861,176.526,24.176,153.884
C04358=1086.168,312.010,412.893,176.523,24.172,153.884
C04359=1086.161,311.763,412.924,176.519,24.167,153.883
C04360=1086.156,311.515,412.956,176.516,24.164,153.883
C04361=1086.150,311.267,412.988,176.513,24.160,153.882
C04362=1086.144,311.020,413.019,176.510,24.156,153.882
C04363=1086.138,310.771,413.050,176.507,24.153,153.881
C04364=1086.133,310.523,413.082,176.504,24.149,153.881
C04365=1086.127,310.275,413.114,176.501,24.145,153.880
C04366=1086.121,310.028,413.145,176.498,24.142,153.880
C04367=1086.115,309.780,413.177,176.495,24.138,153.880
C04368=1086.110,309.532,413.208,176.492,24.134,153.879
C04369=1086.103,309.284,413.240,176.489,24.130,153.879
C04370=1086.098,309.036,413.271,176.486,24.127,153.878
C04371=1086.092,308.787,413.303,176.484,24.123,153.878
C04372=1086.086,308.540,413.334,176.481,24.119,153.877
C04373=1086.080,308.292,413.366,176.478,24.116,153.877
C04374=1086.074,308.044,413.396,176.475,24.112,153.876
C04375=1086.068,307.796,413.428,176.472,24.108,153.876
C04376=1086.063,307.548,413.460,176.469,24.104,153.875
C04377=1086.057,307.300,413.490,176.466,24.101,153.875
C04378=1086.051,307.052,413.522,176.463,24.097,153.875
C04379=1086.046,306.804,413.553,176.460,24.093,153.874
C04380=1086.040,306.557,413.584,176.457,24.090,153.874
C04381=1086.034,306.308,413.615,176.454,24.086,153.873
C04382=1086.028,306.061,413.646,176.451,24.083,153.873
C04383=1086.022,305.812,413.678,176.448,24.078,153.872
C04384=1086.016,305.565,413.709,176.445,24.075,153.872
C04385=1086.011,305.317,413.740,176.442,24.071,153.872
C04386=1086.005,305.069,413.772,176.439,24.067,153.871
C04387=1085.999,304.821,413.802,176.436,24.063,153.871
C04388=1085.994,304.573,413.834,176.433,24.060,153.870
C04389=1085.988,304.325,413.864,176.430,24.056,153.870
C04390=1085.982,304.077,413.896,176.427,24.053,153.869
C04391=1085.973,303.673,413.946,176.422,24.047,153.869
C04392=1085.963,303.269,413.996,176.417,24.040,153.868
C04393=1085.954,302.865,414.047,176.413,24.035,153.867
C04394=1085.945,302.461,414.097,176.408,24.028,153.866
C04395=1085.939,302.213,414.129,176.405,24.025,153.866
C04396=1085.934,301.965,414.160,176.402,24.021,153.866
C04397=1085.928,301.717,414.190,176.399,24.018,153.865
C04398=1085.923,301.469,414.221,176.396,24.014,153.865
C04399=1085.916,301.221,414.252,176.393,24.010,153.864
C04400=1085.911,300.973,414.283,176.391,24.007,153.864
C04401=1085.905,300.725,414.314,176.388,24.003,153.863
C04402=1085.900,300.477,414.345,176.385,24.000,153.863
C04403=1085.894,300.229,414.375,176.382,23.996,153.862
C04404=1085.889,299.982,414.407,176.379,23.992,153.862
C04405=1085.882,299.733,414.437,176.376,23.989,153.862
C04406=1085.877,299.485,414.468,176.373,23.985,153.861
C04407=1085.872,299.237,414.499,176.370,23.981,153.861
C04408=1085.866,298.989,414.529,176.367,23.978,153.860
C04409=1085.861,298.741,414.560,176.364,23.974,153.860
C04410=1085.855,298.493,414.590,176.362,23.970,153.859
C04411=1085.850,298.245,414.621,176.359,23.967,153.859
C04412=1085.843,297.997,414.652,176.356,23.963,153.859
C04413=1085.837,297.749,414.682,176.353,23.960,153.858
C04414=1085.832,297.501,414.713,176.350,23.956,153.858
C04415=1085.827,297.253,414.744,176.347,23.953,153.857
C04416=1085.821,297.005,414.774,176.344,23.949,153.857
C04417=1085.815,296.757,414.804,176.341,23.945,153.857
C04418=1085.809,296.509,414.835,176.338,23.942,153.856
C04419=1085.803,296.261,414.866,176.335,23.938,153.856
C04420=1085.798,296.013,414.896,176.332,23.935,153.855
C04421=1085.792,295.765,414.927,176.330,23.931,153.855
C04422=1085.786,295.517,414.957,176.327,23.928,153.854
C04423=1085.780,295.269,414.987,176.324,23.924,153.854
C04424=1085.775,295.021,415.017,176.321,23.921,153.854
C04425=1085.768,294.772,415.048,176.318,23.918,153.853
C04426=1085.763,294.524,415.079,176.315,23.914,153.853
C04427=1085.757,294.276,415.109,176.312,23.910,153.853
C04428=1085.752,294.028,415.139,176.309,23.907,153.852
C04429=1085.746,293.780,415.169,176.306,23.903,153.852
C04430=1085.740,293.532,415.199,176.303,23.900,153.851
C04431=1085.734,293.285,415.230,176.300,23.896,153.851
C04432=1085.729,293.036,415.259,176.297,23.893,153.851
C04433=1085.723,292.788,415.290,176.295,23.890,153.850
C04434=1085.717,292.540,415.320,176.292,23.886,153.850
C04435=1085.711,292.293,415.351,176.289,23.882,153.849
C04436=1085.706,292.044,415.380,176.286,23.879,153.849
C04437=1085.699,291.796,415.411,176.283,23.876,153.849
C04438=1085.694,291.548,415.441,176.280,23.872,153.848
C04439=1085.688,291.299,415.471,176.277,23.869,153.848
C04440=1085.682,291.052,415.501,176.274,23.865,153.847
C04441=1085.677,290.803,415.531,176.271,23.861,153.847
C04442=1085.671,290.555,415.561,176.269,23.859,153.847
C04443=1085.662,290.165,415.609,176.264,23.853,153.846
C04444=1085.653,289.776,415.656,176.259,23.847,153.846
C04445=1085.645,289.386,415.702,176.255,23.842,153.845
C04446=1085.635,288.995,415.750,176.250,23.837,153.844
C04447=1085.629,288.747,415.780,176.247,23.833,153.844
C04448=1085.624,288.499,415.810,176.244,23.830,153.844
C04449=1085.618,288.251,415.839,176.242,23.827,153.843
C04450=1085.612,288.003,415.869,176.239,23.823,153.843
C04451=1085.606,287.755,415.899,176.236,23.820,153.843
C04452=1085.600,287.507,415.929,176.233,23.816,153.842
C04453=1085.595,287.258,415.959,176.230,23.813,153.842
C04454=1085.589,287.010,415.988,176.227,23.810,153.841
C04455=1085.583,286.762,416.018,176.224,23.806,153.841
C04456=1085.578,286.515,416.047,176.222,23.803,153.841
C04457=1085.572,286.266,416.077,176.219,23.800,153.840
C04458=1085.566,286.018,416.107,176.216,23.796,153.840
C04459=1085.560,285.770,416.136,176.213,23.793,153.839
C04460=1085.555,285.522,416.166,176.210,23.789,153.839
C04461=1085.549,285.274,416.196,176.207,23.786,153.839
C04462=1085.543,285.026,416.226,176.204,23.782,153.838
C04463=1085.537,284.777,416.255,176.202,23.780,153.838
C04464=1085.532,284.529,416.285,176.199,23.776,153.838
C04465=1085.526,284.281,416.314,176.196,23.772,153.837
C04466=1085.520,284.033,416.345,176.193,23.769,153.837
C04467=1085.514,283.785,416.374,176.190,23.766,153.837
C04468=1085.509,283.537,416.403,176.187,23.762,153.836
C04469=1085.504,283.288,416.432,176.185,23.759,153.836
C04470=1085.498,283.040,416.462,176.182,23.756,153.835
C04471=1085.492,282.792,416.491,176.179,23.753,153.835
C04472=1085.486,282.543,416.521,176.176,23.749,153.835
C04473=1085.481,282.296,416.551,176.173,23.745,153.834
C04474=1085.475,282.048,416.580,176.170,23.742,153.834
C04475=1085.469,281.800,416.609,176.168,23.739,153.834
C04476=1085.464,281.551,416.639,176.165,23.735,153.833
C04477=1085.458,281.303,416.668,176.162,23.732,153.833
C04478=1085.452,281.055,416.698,176.159,23.729,153.833
C04479=1085.447,280.806,416.727,176.156,23.726,153.832
C04480=1085.441,280.559,416.756,176.154,23.722,153.832
C04481=1085.435,280.310,416.786,176.150,23.719,153.832
C04482=1085.429,280.062,416.815,176.148,23.716,153.831
C04483=1085.424,279.814,416.844,176.145,23.712,153.831
C04484=1085.417,279.566,416.873,176.142,23.709,153.831
C04485=1085.413,279.317,416.902,176.139,23.706,153.830
C04486=1085.407,279.069,416.931,176.136,23.703,153.830
C04487=1085.401,278.821,416.961,176.133,23.699,153.829
C04488=1085.395,278.573,416.990,176.130,23.696,153.829
C04489=1085.389,278.324,417.019,176.127,23.692,153.829
C04490=1085.384,278.077,417.048,176.125,23.689,153.828
C04491=1085.378,277.828,417.078,176.122,23.686,153.828
C04492=1085.372,277.580,417.106,176.119,23.683,153.828
C04493=1085.367,277.331,417.136,176.116,23.679,153.827
C04494=1085.361,277.084,417.164,176.113,23.676,153.827
C04495=1085.352,276.703,417.209,176.110,23.671,153.826
C04496=1085.343,276.323,417.254,176.105,23.666,153.826
C04497=1085.334,275.943,417.298,176.101,23.661,153.825
C04498=1085.326,275.562,417.342,176.096,23.656,153.825
C04499=1085.320,275.314,417.371,176.093,23.653,153.825
C04500=1085.314,275.066,417.400,176.091,23.650,153.824
C04501=1085.308,274.817,417.429,176.088,23.646,153.824
C04502=1085.303,274.569,417.458,176.085,23.643,153.824
C04503=1085.297,274.321,417.487,176.082,23.639,153.823
C04504=1085.292,274.072,417.516,176.080,23.637,153.823
C04505=1085.286,273.825,417.545,176.077,23.633,153.823
C04506=1085.280,273.576,417.573,176.074,23.630,153.822
C04507=1085.274,273.328,417.602,176.071,23.626,153.822
C04508=1085.269,273.079,417.631,176.069,23.624,153.822
C04509=1085.263,272.831,417.660,176.065,23.620,153.821
C04510=1085.257,272.583,417.689,176.062,23.617,153.821
C04511=1085.252,272.335,417.717,176.059,23.614,153.821
C04512=1085.246,272.087,417.746,176.057,23.610,153.820
C04513=1085.240,271.838,417.775,176.054,23.607,153.820
C04514=1085.235,271.590,417.802,176.051,23.604,153.820
C04515=1085.229,271.342,417.832,176.048,23.601,153.819
C04516=1085.223,271.093,417.860,176.046,23.598,153.819
C04517=1085.218,270.845,417.889,176.043,23.595,153.819
C04518=1085.212,270.596,417.917,176.040,23.591,153.818
C04519=1085.206,270.349,417.946,176.037,23.588,153.818
C04520=1085.200,270.100,417.974,176.035,23.585,153.818
C04521=1085.195,269.851,418.003,176.032,23.582,153.817
C04522=1085.189,269.604,418.032,176.029,23.578,153.817
C04523=1085.183,269.355,418.060,176.026,23.575,153.817
C04524=1085.178,269.107,418.088,176.024,23.572,153.816
C04525=1085.172,268.859,418.117,176.021,23.569,153.816
C04526=1085.166,268.610,418.146,176.018,23.565,153.816
C04527=1085.160,268.362,418.174,176.015,23.563,153.815
C04528=1085.154,268.114,418.203,176.012,23.559,153.815
C04529=1085.149,267.866,418.231,176.009,23.556,153.815
C04530=1085.143,267.617,418.259,176.006,23.553,153.814
C04531=1085.138,267.368,418.288,176.004,23.550,153.814
C04532=1085.132,267.120,418.316,176.001,23.546,153.814
C04533=1085.126,266.872,418.345,175.998,23.543,153.813
C04534=1085.121,266.624,418.373,175.995,23.540,153.813
C04535=1085.115,266.375,418.401,175.993,23.537,153.813
C04536=1085.110,266.127,418.429,175.990,23.534,153.812
C04537=1085.104,265.878,418.457,175.987,23.531,153.812
C04538=1085.098,265.630,418.485,175.985,23.527,153.812
C04539=1085.092,265.382,418.514,175.982,23.524,153.811
C04540=1085.087,265.134,418.542,175.979,23.521,153.811
C04541=1085.081,264.885,418.571,175.977,23.518,153.811
C04542=1085.075,264.637,418.599,175.974,23.515,153.810
C04543=1085.069,264.388,418.627,175.971,23.512,153.810
C04544=1085.064,264.140,418.655,175.968,23.508,153.810
C04545=1085.058,263.892,418.683,175.965,23.505,153.809
C04546=1085.052,263.644,418.711,175.962,23.502,153.809
C04547=1085.043,263.266,418.753,175.958,23.497,153.809
C04548=1085.034,262.888,418.796,175.954,23.493,153.808
C04549=1085.025,262.511,418.839,175.949,23.488,153.808
C04550=1085.016,262.133,418.881,175.946,23.483,153.807
C04551=1085.011,261.885,418.909,175.943,23.480,153.807
C04552=1085.005,261.636,418.937,175.940,23.477,153.807
C04553=1084.999,261.389,418.965,175.937,23.474,153.807
C04554=1084.993,261.140,418.993,175.935,23.471,153.806
C04555=1084.988,260.892,419.021,175.931,23.468,153.806
C04556=1084.982,260.643,419.049,175.929,23.465,153.806
C04557=1084.976,260.395,419.076,175.926,23.462,153.805
C04558=1084.971,260.147,419.104,175.923,23.459,153.805
C04559=1084.965,259.898,419.132,175.921,23.456,153.805
C04560=1084.959,259.650,419.160,175.918,23.452,153.804
C04561=1084.953,259.401,419.188,175.915,23.449,153.804
C04562=1084.948,259.153,419.215,175.913,23.446,153.804
C04563=1084.941,258.904,419.243,175.910,23.443,153.804
C04564=1084.936,258.656,419.271,175.907,23.440,153.803
C04565=1084.930,258.408,419.299,175.904,23.437,153.803
C04566=1084.924,258.159,419.326,175.902,23.434,153.803
C04567=1084.919,257.911,419.354,175.898,23.430,153.802
C04568=1084.913,257.662,419.382,175.896,23.428,153.802
C04569=1084.907,257.414,419.409,175.893,23.425,153.802
C04570=1084.902,257.166,419.437,175.890,23.421,153.801
C04571=1084.896,256.917,419.465,175.888,23.418,153.801
C04572=1084.890,256.669,419.492,175.885,23.415,153.801
C04573=1084.885,256.421,419.520,175.882,23.412,153.801
C04574=1084.879,256.172,419.548,175.880,23.409,153.800
C04575=1084.873,255.924,419.575,175.877,23.406,153.800
C04576=1084.867,255.676,419.603,175.874,23.403,153.800
C04577=1084.861,255.427,419.630,175.872,23.400,153.799
C04578=1084.856,255.179,419.658,175.869,23.396,153.799
C04579=1084.851,254.930,419.685,175.866,23.394,153.799
C04580=1084.844,254.681,419.713,175.863,23.391,153.798
C04581=1084.839,254.433,419.740,175.860,23.387,153.798
C04582=1084.833,254.185,419.767,175.858,23.384,153.798
C04583=1084.827,253.936,419.795,175.855,23.381,153.797
C04584=1084.822,253.688,419.823,175.852,23.378,153.797
C04585=1084.816,253.439,419.849,175.850,23.375,153.797
C04586=1084.811,253.191,419.877,175.847,23.372,153.797
C04587=1084.804,252.942,419.904,175.844,23.368,153.796
C04588=1084.799,252.694,419.932,175.842,23.366,153.796
C04589=1084.793,252.446,419.959,175.839,23.362,153.796
C04590=1084.788,252.197,419.986,175.837,23.360,153.795
C04591=1084.783,251.949,420.014,175.833,23.356,153.795
C04592=1084.777,251.700,420.041,175.831,23.353,153.795
C04593=1084.772,251.451,420.068,175.828,23.350,153.794
C04594=1084.765,251.204,420.096,175.825,23.347,153.794
C04595=1084.760,250.955,420.123,175.823,23.344,153.794
C04596=1084.754,250.706,420.150,175.820,23.340,153.793
C04597=1084.749,250.458,420.178,175.817,23.337,153.793
C04598=1084.743,250.209,420.205,175.815,23.335,153.793
C04599=1084.735,249.829,420.247,175.811,23.330,153.792
C04600=1084.726,249.449,420.288,175.807,23.325,153.792
C04601=1084.718,249.068,420.329,175.802,23.320,153.791
C04602=1084.709,248.688,420.371,175.799,23.315,153.791
C04603=1084.704,248.440,420.398,175.796,23.312,153.791
C04604=1084.698,248.191,420.425,175.794,23.310,153.790
C04605=1084.693,247.943,420.452,175.790,23.306,153.790
C04606=1084.687,247.695,420.479,175.788,23.303,153.790
C04607=1084.682,247.446,420.507,175.785,23.300,153.789
C04608=1084.676,247.197,420.534,175.782,23.297,153.789
C04609=1084.670,246.949,420.560,175.780,23.294,153.789
C04610=1084.665,246.700,420.588,175.777,23.291,153.789
C04611=1084.659,246.452,420.614,175.774,23.287,153.788
C04612=1084.653,246.203,420.641,175.772,23.284,153.788
C04613=1084.648,245.955,420.668,175.769,23.281,153.788
C04614=1084.642,245.706,420.695,175.767,23.279,153.787
C04615=1084.636,245.457,420.722,175.764,23.275,153.787
C04616=1084.630,245.209,420.748,175.762,23.273,153.787
C04617=1084.625,244.960,420.776,175.759,23.269,153.787
C04618=1084.619,244.712,420.802,175.756,23.266,153.786
C04619=1084.614,244.464,420.829,175.753,23.263,153.786
C04620=1084.609,244.215,420.856,175.750,23.260,153.786
C04621=1084.603,243.967,420.883,175.748,23.257,153.785
C04622=1084.597,243.718,420.910,175.745,23.254,153.785
C04623=1084.591,243.470,420.936,175.743,23.251,153.785
C04624=1084.585,243.221,420.963,175.740,23.248,153.784
C04625=1084.580,242.973,420.990,175.737,23.244,153.784
C04626=1084.575,242.724,421.017,175.735,23.242,153.784
C04627=1084.569,242.476,421.043,175.732,23.238,153.784
C04628=1084.563,242.226,421.070,175.730,23.236,153.783
C04629=1084.557,241.978,421.096,175.727,23.232,153.783
C04630=1084.551,241.730,421.123,175.724,23.230,153.783
C04631=1084.546,241.481,421.150,175.721,23.227,153.782
C04632=1084.540,241.233,421.176,175.719,23.224,153.782
C04633=1084.534,240.984,421.202,175.716,23.221,153.782
C04634=1084.528,240.736,421.229,175.713,23.217,153.782
C04635=1084.523,240.487,421.255,175.711,23.215,153.781
C04636=1084.517,240.239,421.282,175.708,23.211,153.781
C04637=1084.511,239.990,421.308,175.706,23.209,153.781
C04638=1084.506,239.741,421.335,175.703,23.206,153.780
C04639=1084.501,239.493,421.362,175.701,23.203,153.780
C04640=1084.494,239.245,421.388,175.697,23.200,153.780
C04641=1084.489,238.996,421.414,175.695,23.197,153.780
C04642=1084.483,238.747,421.441,175.692,23.194,153.779
C04643=1084.477,238.499,421.467,175.690,23.190,153.779
C04644=1084.472,238.250,421.493,175.687,23.187,153.779
C04645=1084.466,238.002,421.520,175.685,23.184,153.778
C04646=1084.460,237.753,421.546,175.682,23.181,153.778
C04647=1084.455,237.504,421.572,175.680,23.179,153.778
C04648=1084.449,237.256,421.599,175.677,23.175,153.778
C04649=1084.443,237.007,421.625,175.675,23.173,153.777
C04650=1084.438,236.759,421.652,175.672,23.169,153.777
C04651=1084.429,236.372,421.692,175.668,23.165,153.777
C04652=1084.420,235.985,421.733,175.664,23.160,153.776
C04653=1084.411,235.598,421.774,175.660,23.156,153.776
C04654=1084.402,235.210,421.815,175.655,23.151,153.775
C04655=1084.397,234.961,421.841,175.653,23.148,153.775
C04656=1084.391,234.713,421.867,175.650,23.145,153.775
C04657=1084.386,234.465,421.893,175.648,23.142,153.774
C04658=1084.381,234.216,421.920,175.645,23.138,153.774
C04659=1084.375,233.967,421.946,175.643,23.136,153.774
C04660=1084.369,233.719,421.972,175.640,23.132,153.773
C04661=1084.363,233.470,421.998,175.638,23.130,153.773
C04662=1084.358,233.221,422.023,175.635,23.126,153.773
C04663=1084.352,232.973,422.050,175.632,23.124,153.773
C04664=1084.346,232.724,422.076,175.629,23.120,153.772
C04665=1084.342,232.476,422.102,175.627,23.118,153.772
C04666=1084.335,232.228,422.128,175.624,23.114,153.772
C04667=1084.330,231.979,422.154,175.622,23.112,153.772
C04668=1084.324,231.730,422.180,175.619,23.109,153.771
C04669=1084.318,231.481,422.206,175.617,23.106,153.771
C04670=1084.313,231.232,422.232,175.614,23.103,153.771
C04671=1084.307,230.984,422.257,175.612,23.100,153.770
C04672=1084.302,230.735,422.283,175.609,23.097,153.770
C04673=1084.296,230.487,422.310,175.606,23.094,153.770
C04674=1084.290,230.238,422.335,175.604,23.090,153.769
C04675=1084.284,229.989,422.361,175.601,23.087,153.769
C04676=1084.279,229.740,422.387,175.598,23.085,153.769
C04677=1084.273,229.492,422.412,175.596,23.082,153.769
C04678=1084.268,229.244,422.439,175.593,23.079,153.769
C04679=1084.261,228.995,422.464,175.591,23.076,153.768
C04680=1084.256,228.746,422.490,175.589,23.073,153.768
C04681=1084.250,228.497,422.516,175.586,23.070,153.768
C04682=1084.245,228.250,422.541,175.584,23.067,153.767
C04683=1084.239,228.001,422.567,175.580,23.064,153.767
C04684=1084.233,227.752,422.592,175.578,23.061,153.767
C04685=1084.228,227.503,422.618,175.575,23.058,153.767
C04686=1084.222,227.255,422.645,175.573,23.055,153.766
C04687=1084.216,227.007,422.670,175.570,23.052,153.766
C04688=1084.211,226.758,422.695,175.568,23.049,153.766
C04689=1084.205,226.509,422.721,175.565,23.046,153.765
C04690=1084.199,226.260,422.747,175.563,23.043,153.765
C04691=1084.194,226.012,422.772,175.561,23.040,153.765
C04692=1084.188,225.763,422.798,175.558,23.037,153.764
C04693=1084.182,225.514,422.823,175.556,23.034,153.764
C04694=1084.176,225.265,422.849,175.553,23.031,153.764
C04695=1084.171,225.017,422.874,175.550,23.028,153.764
C04696=1084.165,224.768,422.900,175.547,23.025,153.763
C04697=1084.159,224.520,422.925,175.545,23.022,153.763
C04698=1084.155,224.271,422.950,175.542,23.019,153.763
C04699=1084.148,224.022,422.975,175.540,23.016,153.763
C04700=1084.143,223.773,423.001,175.538,23.013,153.762
C04701=1084.137,223.525,423.026,175.535,23.010,153.762
C04702=1084.132,223.276,423.052,175.533,23.007,153.762
C04703=1084.123,222.880,423.092,175.528,23.002,153.761
C04704=1084.114,222.485,423.133,175.525,22.998,153.761
C04705=1084.105,222.089,423.173,175.520,22.993,153.760
C04706=1084.096,221.693,423.213,175.516,22.989,153.760
C04707=1084.090,221.445,423.238,175.513,22.985,153.760
C04708=1084.085,221.197,423.264,175.511,22.983,153.759
C04709=1084.079,220.948,423.289,175.509,22.980,153.759
C04710=1084.073,220.699,423.314,175.506,22.977,153.759
C04711=1084.068,220.450,423.340,175.504,22.974,153.759
C04712=1084.062,220.202,423.365,175.501,22.971,153.758
C04713=1084.056,219.953,423.390,175.499,22.968,153.758
C04714=1084.050,219.704,423.414,175.497,22.965,153.758
C04715=1084.045,219.455,423.440,175.494,22.962,153.758
C04716=1084.039,219.207,423.466,175.491,22.959,153.757
C04717=1084.033,218.958,423.490,175.488,22.956,153.757
C04718=1084.027,218.709,423.515,175.486,22.953,153.757
C04719=1084.022,218.461,423.541,175.484,22.950,153.756
C04720=1084.016,218.212,423.566,175.481,22.947,153.756
C04721=1084.011,217.964,423.590,175.479,22.944,153.756
C04722=1084.005,217.715,423.615,175.476,22.941,153.756
C04723=1083.999,217.466,423.641,175.474,22.938,153.755
C04724=1083.994,217.218,423.666,175.472,22.936,153.755
C04725=1083.988,216.968,423.691,175.469,22.932,153.755
C04726=1083.982,216.720,423.716,175.467,22.930,153.754
C04727=1083.977,216.471,423.741,175.464,22.926,153.754
C04728=1083.971,216.223,423.766,175.461,22.924,153.754
C04729=1083.966,215.974,423.790,175.459,22.921,153.754
C04730=1083.960,215.726,423.815,175.456,22.918,153.753
C04731=1083.954,215.476,423.840,175.454,22.915,153.753
C04732=1083.948,215.228,423.865,175.452,22.912,153.753
C04733=1083.943,214.979,423.890,175.449,22.909,153.753
C04734=1083.938,214.731,423.915,175.447,22.906,153.752
C04735=1083.932,214.481,423.940,175.444,22.903,153.752
C04736=1083.926,214.233,423.964,175.442,22.900,153.752
C04737=1083.920,213.984,423.989,175.440,22.897,153.751
C04738=1083.916,213.735,424.014,175.437,22.894,153.751
C04739=1083.909,213.487,424.040,175.434,22.891,153.751
C04740=1083.904,213.238,424.064,175.432,22.888,153.750
C04741=1083.898,212.989,424.088,175.429,22.885,153.750
C04742=1083.893,212.741,424.113,175.427,22.882,153.750
C04743=1083.887,212.492,424.138,175.424,22.879,153.750
C04744=1083.881,212.243,424.162,175.422,22.876,153.749
C04745=1083.875,211.994,424.188,175.420,22.873,153.749
C04746=1083.870,211.746,424.212,175.417,22.870,153.749
C04747=1083.864,211.496,424.237,175.415,22.867,153.749
C04748=1083.859,211.248,424.261,175.413,22.864,153.748
C04749=1083.853,211.000,424.286,175.410,22.861,153.748
C04750=1083.847,210.751,424.310,175.407,22.858,153.748
C04751=1083.842,210.502,424.335,175.405,22.856,153.747
C04752=1083.836,210.253,424.359,175.402,22.852,153.747
C04753=1083.830,210.005,424.384,175.400,22.850,153.747
C04754=1083.825,209.755,424.409,175.398,22.847,153.747
C04755=1083.816,209.364,424.447,175.393,22.842,153.746
C04756=1083.807,208.972,424.486,175.390,22.838,153.746
C04757=1083.798,208.581,424.524,175.386,22.833,153.745
C04758=1083.789,208.189,424.563,175.382,22.828,153.745
C04759=1083.766,207.159,424.662,175.294,22.782,153.748
C04760=1083.761,206.910,424.686,175.292,22.780,153.748
C04761=1083.755,206.662,424.710,175.289,22.778,153.748
C04762=1083.749,206.412,424.734,175.287,22.776,153.747
C04763=1083.744,206.164,424.758,175.284,22.774,153.747
C04764=1083.738,205.915,424.782,175.282,22.772,153.747
C04765=1083.733,205.666,424.805,175.279,22.770,153.747
C04766=1083.727,205.418,424.829,175.276,22.768,153.747
C04767=1083.721,205.169,424.853,175.274,22.766,153.747
C04768=1083.716,204.919,424.877,175.271,22.764,153.747
C04769=1083.710,204.671,424.901,175.269,22.762,153.747
C04770=1083.704,204.423,424.925,175.267,22.760,153.747
C04771=1083.699,204.173,424.949,175.264,22.758,153.747
C04772=1083.693,203.925,424.972,175.262,22.756,153.747
C04773=1083.688,203.676,424.997,175.258,22.754,153.747
C04774=1083.682,203.428,425.019,175.256,22.752,153.747
C04775=1083.676,203.178,425.044,175.254,22.750,153.747
C04776=1083.671,202.929,425.068,175.251,22.748,153.747
C04777=1083.665,202.681,425.091,175.249,22.746,153.747
C04778=1083.660,202.432,425.115,175.246,22.744,153.746
C04779=1083.654,202.183,425.138,175.244,22.742,153.746
C04780=1083.649,201.934,425.162,175.241,22.740,153.746
C04781=1083.643,201.686,425.186,175.239,22.738,153.746
C04782=1083.637,201.436,425.209,175.236,22.736,153.746
C04783=1083.632,201.188,425.233,175.233,22.734,153.746
C04784=1083.626,200.939,425.256,175.231,22.732,153.746
C04785=1083.620,200.690,425.280,175.228,22.730,153.746
C04786=1083.615,200.441,425.303,175.226,22.728,153.746
C04787=1083.609,200.193,425.327,175.223,22.726,153.746
C04788=1083.604,199.944,425.351,175.221,22.725,153.746
C04789=1083.597,199.695,425.375,175.218,22.723,153.746
C04790=1083.591,199.446,425.398,175.216,22.720,153.746
C04791=1083.586,199.197,425.422,175.214,22.719,153.746
C04792=1083.580,198.948,425.445,175.211,22.717,153.746
C04793=1083.575,198.700,425.468,175.209,22.715,153.746
C04794=1083.569,198.451,425.492,175.206,22.713,153.746
C04795=1083.564,198.202,425.515,175.203,22.711,153.746
C04796=1083.558,197.953,425.538,175.200,22.709,153.746
C04797=1083.553,197.705,425.562,175.198,22.707,153.746
C04798=1083.547,197.456,425.585,175.196,22.705,153.746
C04799=1083.541,197.207,425.608,175.193,22.703,153.745
C04800=1083.536,196.958,425.632,175.191,22.701,153.745
C04801=1083.530,196.709,425.656,175.188,22.699,153.745
C04802=1083.524,196.460,425.679,175.186,22.697,153.745
C04803=1083.518,196.211,425.701,175.183,22.695,153.745
C04804=1083.513,195.962,425.726,175.181,22.693,153.745
C04805=1083.507,195.713,425.749,175.179,22.691,153.745
C04806=1083.501,195.464,425.772,175.176,22.689,153.745
C04807=1083.496,195.215,425.795,175.174,22.688,153.745
C04808=1083.490,194.967,425.819,175.171,22.685,153.745
C04809=1083.485,194.718,425.842,175.169,22.684,153.745
C04810=1083.479,194.469,425.865,175.166,22.682,153.745
C04811=1083.474,194.220,425.888,175.164,22.680,153.745
C04812=1083.468,193.971,425.911,175.162,22.678,153.745
C04813=1083.462,193.723,425.935,175.158,22.676,153.745
C04814=1083.456,193.474,425.958,175.156,22.673,153.745
C04815=1083.451,193.225,425.981,175.153,22.671,153.745
C04816=1083.446,192.976,426.004,175.151,22.670,153.745
C04817=1083.441,192.728,426.027,175.149,22.667,153.744
C04818=1083.435,192.479,426.050,175.146,22.666,153.744
C04819=1083.430,192.229,426.073,175.144,22.663,153.744
C04820=1083.423,191.951,426.099,175.141,22.662,153.744
C04821=1083.416,191.672,426.125,175.139,22.659,153.744
C04822=1083.411,191.394,426.151,175.136,22.657,153.744
C04823=1083.404,191.114,426.177,175.133,22.655,153.744
C04824=1083.399,190.865,426.200,175.131,22.653,153.744
C04825=1083.393,190.616,426.223,175.128,22.651,153.744
C04826=1083.388,190.367,426.246,175.126,22.649,153.744
C04827=1083.383,190.119,426.269,175.124,22.647,153.744
C04828=1083.377,189.870,426.292,175.121,22.645,153.744
C04829=1083.371,189.621,426.315,175.119,22.643,153.744
C04830=1083.366,189.372,426.338,175.116,22.641,153.744
C04831=1083.361,189.123,426.361,175.114,22.639,153.743
C04832=1083.355,188.874,426.384,175.112,22.637,153.743
C04833=1083.349,188.625,426.407,175.109,22.635,153.743
C04834=1083.344,188.377,426.430,175.107,22.633,153.743
C04835=1083.338,188.128,426.453,175.104,22.631,153.743
C04836=1083.333,187.879,426.476,175.102,22.629,153.743
C04837=1083.328,187.630,426.499,175.100,22.627,153.743
C04838=1083.322,187.381,426.522,175.097,22.625,153.743
C04839=1083.316,187.132,426.544,175.095,22.623,153.743
C04840=1083.311,186.883,426.567,175.092,22.621,153.743
C04841=1083.306,186.635,426.590,175.090,22.619,153.743
C04842=1083.300,186.386,426.613,175.087,22.617,153.743
C04843=1083.294,186.137,426.636,175.085,22.615,153.743
C04844=1083.290,185.888,426.659,175.083,22.613,153.743
C04845=1083.284,185.639,426.681,175.080,22.611,153.742
C04846=1083.279,185.390,426.704,175.078,22.609,153.742
C04847=1083.273,185.141,426.727,175.076,22.607,153.742
C04848=1083.267,184.892,426.750,175.073,22.605,153.742
C04849=1083.262,184.642,426.772,175.071,22.603,153.742
C04850=1083.256,184.395,426.794,175.068,22.601,153.742
C04851=1083.250,184.146,426.817,175.066,22.599,153.742
C04852=1083.244,183.897,426.840,175.063,22.597,153.742
C04853=1083.239,183.647,426.862,175.061,22.595,153.742
C04854=1083.233,183.398,426.885,175.058,22.594,153.742
C04855=1083.227,183.150,426.908,175.056,22.591,153.742
C04856=1083.221,182.900,426.930,175.054,22.590,153.742
C04857=1083.216,182.651,426.953,175.051,22.588,153.742
C04858=1083.210,182.403,426.975,175.049,22.586,153.742
C04859=1083.204,182.154,426.997,175.047,22.584,153.742
C04860=1083.199,181.905,427.020,175.045,22.582,153.742
C04861=1083.193,181.656,427.043,175.042,22.581,153.742
C04862=1083.187,181.407,427.065,175.040,22.579,153.742
C04863=1083.181,181.158,427.088,175.038,22.576,153.741
C04864=1083.176,180.910,427.110,175.035,22.575,153.741
C04865=1083.170,180.660,427.132,175.033,22.573,153.741
C04866=1083.164,180.412,427.155,175.030,22.571,153.741
C04867=1083.159,180.162,427.177,175.028,22.569,153.741
C04868=1083.153,179.913,427.200,175.025,22.567,153.741
C04869=1083.147,179.665,427.221,175.023,22.565,153.741
C04870=1083.141,179.416,427.244,175.021,22.563,153.741
C04871=1083.136,179.167,427.267,175.018,22.561,153.741
C04872=1083.130,178.918,427.289,175.016,22.559,153.741
C04873=1083.124,178.670,427.311,175.013,22.557,153.741
C04874=1083.119,178.420,427.333,175.012,22.556,153.741
C04875=1083.113,178.171,427.356,175.009,22.554,153.741
C04876=1083.107,177.922,427.378,175.007,22.552,153.741
C04877=1083.102,177.673,427.400,175.004,22.550,153.741
C04878=1083.097,177.424,427.423,175.002,22.548,153.741
C04879=1083.090,177.175,427.444,175.000,22.546,153.741
C04880=1083.085,176.926,427.467,174.997,22.544,153.741
C04881=1083.080,176.677,427.489,174.995,22.542,153.741
C04882=1083.073,176.429,427.512,174.992,22.540,153.740
C04883=1083.068,176.179,427.534,174.990,22.538,153.740
C04884=1083.062,175.901,427.559,174.988,22.536,153.740
C04885=1083.055,175.621,427.583,174.985,22.534,153.740
C04886=1083.050,175.343,427.609,174.983,22.532,153.740
C04887=1083.043,175.063,427.633,174.979,22.529,153.740
C04888=1083.037,174.814,427.656,174.978,22.527,153.740
C04889=1083.032,174.565,427.677,174.976,22.526,153.740
C04890=1083.026,174.316,427.699,174.973,22.524,153.740
C04891=1083.020,174.067,427.722,174.971,22.522,153.740
C04892=1083.015,173.819,427.744,174.968,22.520,153.740
C04893=1083.010,173.569,427.766,174.966,22.517,153.740
C04894=1083.004,173.321,427.787,174.964,22.516,153.740
C04895=1082.998,173.072,427.810,174.961,22.514,153.740
C04896=1082.992,172.822,427.832,174.959,22.512,153.739
C04897=1082.987,172.574,427.854,174.957,22.510,153.739
C04898=1082.982,172.324,427.876,174.955,22.508,153.739
C04899=1082.975,172.075,427.898,174.952,22.506,153.739
C04900=1082.971,171.827,427.920,174.950,22.504,153.739
C04901=1082.964,171.577,427.942,174.948,22.502,153.739
C04902=1082.960,171.329,427.964,174.945,22.500,153.739
C04903=1082.953,171.079,427.985,174.943,22.498,153.739
C04904=1082.948,170.831,428.008,174.940,22.496,153.739
C04905=1082.943,170.582,428.030,174.939,22.494,153.739
C04906=1082.937,170.333,428.052,174.937,22.492,153.739
C04907=1082.932,170.084,428.073,174.934,22.490,153.739
C04908=1082.926,169.834,428.095,174.932,22.488,153.739
C04909=1082.921,169.586,428.117,174.929,22.486,153.738
C04910=1082.915,169.336,428.139,174.927,22.484,153.738
C04911=1082.910,169.088,428.161,174.925,22.482,153.738
C04912=1082.903,168.839,428.183,174.923,22.481,153.738
C04913=1082.899,168.590,428.205,174.921,22.478,153.738
C04914=1082.892,168.341,428.226,174.918,22.476,153.738
C04915=1082.888,168.092,428.248,174.916,22.474,153.738
C04916=1082.881,167.843,428.270,174.914,22.472,153.738
C04917=1082.877,167.594,428.292,174.911,22.470,153.738
C04918=1082.870,167.345,428.313,174.910,22.469,153.738
C04919=1082.866,167.096,428.335,174.907,22.466,153.738
C04920=1082.859,166.847,428.357,174.905,22.465,153.738
C04921=1082.855,166.598,428.379,174.903,22.462,153.737
C04922=1082.848,166.349,428.400,174.900,22.460,153.737
C04923=1082.844,166.100,428.422,174.898,22.458,153.737
C04924=1082.837,165.851,428.444,174.897,22.456,153.737
C04925=1082.833,165.602,428.466,174.894,22.454,153.737
C04926=1082.827,165.353,428.487,174.892,22.452,153.737
C04927=1082.822,165.104,428.509,174.889,22.450,153.737
C04928=1082.816,164.855,428.531,174.887,22.448,153.737
C04929=1082.811,164.606,428.553,174.885,22.446,153.737
C04930=1082.805,164.358,428.574,174.883,22.444,153.737
C04931=1082.800,164.107,428.595,174.881,22.442,153.736
C04932=1082.794,163.859,428.617,174.878,22.440,153.736
C04933=1082.789,163.609,428.639,174.876,22.438,153.736
C04934=1082.783,163.361,428.660,174.874,22.436,153.736
C04935=1082.778,163.112,428.682,174.872,22.434,153.736
C04936=1082.772,162.863,428.704,174.870,22.432,153.736
C04937=1082.767,162.614,428.725,174.867,22.430,153.736
C04938=1082.762,162.364,428.747,174.865,22.428,153.736
C04939=1082.756,162.116,428.768,174.863,22.426,153.736
C04940=1082.751,161.867,428.790,174.860,22.424,153.736
C04941=1082.745,161.618,428.811,174.859,22.422,153.735
C04942=1082.740,161.369,428.833,174.856,22.420,153.735
C04943=1082.735,161.119,428.854,174.854,22.418,153.735
C04944=1082.729,160.871,428.875,174.852,22.416,153.735
C04945=1082.723,160.622,428.897,174.849,22.414,153.735
C04946=1082.717,160.373,428.918,174.848,22.412,153.735
C04947=1082.712,160.124,428.939,174.846,22.410,153.735
C04948=1082.705,159.844,428.963,174.843,22.408,153.735
C04949=1082.699,159.565,428.987,174.841,22.406,153.735
C04950=1082.693,159.285,429.011,174.838,22.403,153.735
C04951=1082.686,159.006,429.035,174.835,22.401,153.735
C04952=1082.681,158.756,429.057,174.834,22.399,153.734
C04953=1082.676,158.507,429.077,174.831,22.398,153.734
C04954=1082.670,158.259,429.099,174.829,22.395,153.734
C04955=1082.664,158.010,429.120,174.827,22.393,153.734
C04956=1082.659,157.761,429.141,174.824,22.391,153.734
C04957=1082.653,157.511,429.162,174.823,22.390,153.734
C04958=1082.647,157.263,429.184,174.820,22.387,153.734
C04959=1082.642,157.014,429.204,174.818,22.385,153.734
C04960=1082.636,156.764,429.227,174.816,22.383,153.734
C04961=1082.631,156.516,429.248,174.814,22.381,153.734
C04962=1082.626,156.267,429.268,174.812,22.380,153.734
C04963=1082.619,156.017,429.290,174.809,22.377,153.734
C04964=1082.614,155.768,429.311,174.807,22.376,153.734
C04965=1082.609,155.520,429.332,174.806,22.374,153.733
C04966=1082.603,155.270,429.353,174.803,22.372,153.733
C04967=1082.597,155.021,429.374,174.801,22.370,153.733
C04968=1082.591,154.772,429.395,174.798,22.368,153.733
C04969=1082.586,154.523,429.416,174.797,22.366,153.733
C04970=1082.581,154.274,429.437,174.795,22.364,153.733
C04971=1082.574,154.025,429.458,174.792,22.362,153.733
C04972=1082.569,153.776,429.479,174.790,22.359,153.733
C04973=1082.564,153.527,429.500,174.788,22.358,153.733
C04974=1082.558,153.277,429.521,174.786,22.356,153.733
C04975=1082.552,153.029,429.542,174.784,22.354,153.732
C04976=1082.547,152.780,429.563,174.781,22.352,153.732
C04977=1082.541,152.531,429.584,174.780,22.350,153.732
C04978=1082.535,152.281,429.605,174.777,22.348,153.732
C04979=1082.530,152.032,429.626,174.775,22.346,153.732
C04980=1082.525,151.784,429.647,174.773,22.344,153.732
C04981=1082.519,151.534,429.668,174.771,22.342,153.732
C04982=1082.513,151.285,429.689,174.769,22.340,153.732
C04983=1082.508,151.036,429.710,174.767,22.338,153.732
C04984=1082.502,150.787,429.730,174.764,22.335,153.732
C04985=1082.496,150.538,429.751,174.763,22.334,153.731
C04986=1082.491,150.289,429.772,174.760,22.332,153.731
C04987=1082.485,150.040,429.792,174.758,22.329,153.731
C04988=1082.480,149.791,429.814,174.756,22.328,153.731
C04989=1082.474,149.542,429.835,174.754,22.326,153.731
C04990=1082.469,149.293,429.855,174.752,22.324,153.731
C04991=1082.463,149.044,429.876,174.750,22.322,153.731
C04992=1082.458,148.795,429.897,174.748,22.320,153.731
C04993=1082.451,148.545,429.917,174.746,22.318,153.731
C04994=1082.446,148.296,429.938,174.743,22.316,153.731
C04995=1082.440,148.048,429.959,174.741,22.314,153.731
C04996=1082.435,147.799,429.980,174.739,22.312,153.730
C04997=1082.429,147.549,430.001,174.737,22.310,153.730
C04998=1082.423,147.300,430.021,174.735,22.308,153.730
C04999=1082.418,147.051,430.042,174.733,22.306,153.730
C05000=1082.412,146.802,430.062,174.731,22.304,153.730
C05001=1082.407,146.553,430.083,174.729,22.302,153.730
C05002=1082.401,146.304,430.103,174.726,22.299,153.730
C05003=1082.395,146.055,430.124,174.725,22.298,153.730
C05004=1082.390,145.806,430.145,174.722,22.296,153.730
C05005=1082.383,145.557,430.165,174.720,22.294,153.730
C05006=1082.378,145.307,430.186,174.719,22.292,153.729
C05007=1082.373,145.058,430.206,174.716,22.290,153.729
C05008=1082.367,144.809,430.227,174.714,22.288,153.729
C05009=1082.361,144.560,430.247,174.712,22.286,153.729
C05010=1082.356,144.311,430.268,174.710,22.284,153.729
C05011=1082.350,144.061,430.288,174.708,22.282,153.729
C05012=1082.344,143.782,430.311,174.705,22.280,153.729
C05013=1082.337,143.503,430.334,174.703,22.277,153.729
C05014=1082.331,143.222,430.358,174.701,22.275,153.728
C05015=1082.325,142.943,430.381,174.699,22.273,153.728
C05016=1082.320,142.694,430.401,174.696,22.271,153.728
C05017=1082.314,142.445,430.422,174.695,22.269,153.728
C05018=1082.308,142.196,430.442,174.692,22.267,153.728
C05019=1082.303,141.947,430.462,174.690,22.264,153.728
C05020=1082.297,141.697,430.483,174.689,22.263,153.728
C05021=1082.291,141.448,430.503,174.686,22.261,153.728
C05022=1082.286,141.199,430.524,174.684,22.258,153.728
C05023=1082.281,140.950,430.544,174.682,22.257,153.728
C05024=1082.275,140.701,430.564,174.680,22.254,153.727
C05025=1082.269,140.452,430.585,174.678,22.252,153.727
C05026=1082.263,140.203,430.605,174.677,22.250,153.727
C05027=1082.258,139.954,430.625,174.674,22.248,153.727
C05028=1082.252,139.705,430.645,174.672,22.246,153.727
C05029=1082.246,139.456,430.666,174.670,22.244,153.727
C05030=1082.241,139.206,430.687,174.668,22.242,153.727
C05031=1082.235,138.958,430.707,174.666,22.240,153.727
C05032=1082.230,138.708,430.726,174.664,22.238,153.726
C05033=1082.224,138.459,430.746,174.662,22.236,153.726
C05034=1082.219,138.210,430.767,174.660,22.234,153.726
C05035=1082.213,137.961,430.787,174.658,22.232,153.726
C05036=1082.208,137.712,430.807,174.656,22.230,153.726
C05037=1082.202,137.463,430.827,174.653,22.228,153.726
C05038=1082.196,137.214,430.848,174.652,22.226,153.726
C05039=1082.190,136.964,430.868,174.650,22.224,153.726
C05040=1082.185,136.715,430.888,174.647,22.222,153.726
C05041=1082.179,136.466,430.908,174.646,22.220,153.725
C05042=1082.173,136.217,430.928,174.644,22.218,153.725
C05043=1082.168,135.968,430.949,174.641,22.215,153.725
C05044=1082.162,135.719,430.968,174.640,22.214,153.725
C05045=1082.157,135.469,430.988,174.637,22.212,153.725
C05046=1082.151,135.221,431.008,174.635,22.209,153.725
C05047=1082.145,134.972,431.029,174.634,22.208,153.725
C05048=1082.140,134.722,431.048,174.631,22.206,153.725
C05049=1082.134,134.473,431.069,174.629,22.203,153.725
C05050=1082.128,134.224,431.089,174.628,22.201,153.724
C05051=1082.122,133.975,431.109,174.625,22.199,153.724
C05052=1082.118,133.726,431.128,174.624,22.198,153.724
C05053=1082.112,133.477,431.148,174.622,22.195,153.724
C05054=1082.106,133.228,431.169,174.619,22.193,153.724
C05055=1082.101,132.978,431.188,174.618,22.191,153.724
C05056=1082.095,132.729,431.208,174.615,22.189,153.724
C05057=1082.089,132.480,431.229,174.613,22.187,153.724
C05058=1082.084,132.231,431.248,174.612,22.185,153.723
C05059=1082.078,131.982,431.269,174.610,22.183,153.723
C05060=1082.072,131.733,431.288,174.607,22.180,153.723
C05061=1082.067,131.484,431.308,174.606,22.179,153.723
C05062=1082.061,131.235,431.328,174.603,22.177,153.723
C05063=1082.055,130.985,431.347,174.602,22.175,153.723
C05064=1082.050,130.736,431.367,174.600,22.173,153.723
C05065=1082.044,130.487,431.387,174.597,22.171,153.723
C05066=1082.038,130.238,431.407,174.596,22.169,153.722
C05067=1082.032,129.989,431.427,174.594,22.166,153.722
C05068=1082.026,129.740,431.446,174.592,22.165,153.722
C05069=1082.020,129.491,431.466,174.590,22.163,153.722
C05070=1082.015,129.241,431.486,174.587,22.160,153.722
C05071=1082.009,128.992,431.506,174.586,22.159,153.722
C05072=1082.004,128.743,431.525,174.584,22.157,153.722
C05073=1081.998,128.494,431.545,174.581,22.154,153.722
C05074=1081.992,128.245,431.564,174.580,22.153,153.721
C05075=1081.986,127.996,431.584,174.578,22.150,153.721
C05076=1081.980,127.716,431.606,174.575,22.148,153.721
C05077=1081.973,127.435,431.629,174.573,22.145,153.721
C05078=1081.967,127.155,431.651,174.572,22.144,153.721
C05079=1081.961,126.876,431.673,174.570,22.141,153.721
C05080=1081.955,126.626,431.693,174.567,22.139,153.721
C05081=1081.949,126.377,431.712,174.565,22.137,153.721
C05082=1081.943,126.128,431.732,174.563,22.135,153.720
C05083=1081.938,125.879,431.751,174.561,22.133,153.720
C05084=1081.932,125.631,431.771,174.560,22.131,153.720
C05085=1081.927,125.381,431.790,174.557,22.129,153.720
C05086=1081.921,125.132,431.809,174.555,22.127,153.720
C05087=1081.916,124.883,431.830,174.554,22.125,153.720
C05088=1081.910,124.633,431.849,174.551,22.123,153.720
C05089=1081.904,124.384,431.868,174.550,22.121,153.719
C05090=1081.898,124.135,431.888,174.548,22.118,153.719
C05091=1081.893,123.886,431.907,174.545,22.116,153.719
C05092=1081.887,123.636,431.927,174.544,22.115,153.719
C05093=1081.882,123.388,431.946,174.542,22.112,153.719
C05094=1081.876,123.139,431.965,174.540,22.110,153.719
C05095=1081.870,122.889,431.985,174.538,22.108,153.719
C05096=1081.864,122.640,432.005,174.537,22.106,153.719
C05097=1081.858,122.391,432.024,174.534,22.104,153.718
C05098=1081.854,122.141,432.044,174.532,22.101,153.718
C05099=1081.848,121.892,432.063,174.531,22.100,153.718
C05100=1081.842,121.644,432.083,174.528,22.098,153.718
C05101=1081.837,121.394,432.102,174.527,22.096,153.718
C05102=1081.831,121.145,432.121,174.525,22.094,153.718
C05103=1081.825,120.895,432.140,174.523,22.092,153.718
C05104=1081.819,120.647,432.160,174.521,22.089,153.717
C05105=1081.814,120.397,432.180,174.519,22.087,153.717
C05106=1081.809,120.148,432.198,174.517,22.085,153.717
C05107=1081.803,119.899,432.218,174.515,22.083,153.717
C05108=1081.797,119.650,432.237,174.514,22.081,153.717
C05109=1081.791,119.401,432.257,174.511,22.078,153.717
C05110=1081.786,119.151,432.276,174.510,22.077,153.717
C05111=1081.780,118.903,432.295,174.508,22.074,153.716
C05112=1081.775,118.653,432.314,174.505,22.072,153.716
C05113=1081.769,118.404,432.333,174.504,22.070,153.716
C05114=1081.763,118.154,432.353,174.502,22.068,153.716
C05115=1081.758,117.906,432.372,174.500,22.066,153.716
C05116=1081.752,117.657,432.392,174.498,22.063,153.716
C05117=1081.747,117.407,432.411,174.497,22.061,153.715
C05118=1081.741,117.158,432.430,174.494,22.059,153.715
C05119=1081.736,116.909,432.449,174.493,22.057,153.715
C05120=1081.730,116.660,432.468,174.491,22.055,153.715
C05121=1081.725,116.410,432.487,174.489,22.053,153.715
C05122=1081.719,116.161,432.507,174.487,22.051,153.715
C05123=1081.714,115.912,432.525,174.485,22.048,153.715
C05124=1081.708,115.663,432.545,174.484,22.046,153.714
C05125=1081.702,115.413,432.564,174.481,22.044,153.714
C05126=1081.697,115.164,432.583,174.480,22.042,153.714
C05127=1081.692,114.915,432.602,174.478,22.040,153.714
C05128=1081.686,114.666,432.621,174.476,22.038,153.714
C05129=1081.681,114.417,432.640,174.474,22.036,153.714
C05130=1081.675,114.167,432.659,174.472,22.033,153.713
C05131=1081.669,113.918,432.679,174.470,22.031,153.713
C05132=1081.663,113.669,432.697,174.468,22.029,153.713
C05133=1081.658,113.420,432.716,174.467,22.027,153.713
C05134=1081.652,113.171,432.735,174.464,22.025,153.713
C05135=1081.647,112.921,432.755,174.463,22.023,153.713
C05136=1081.641,112.672,432.774,174.461,22.020,153.713
C05137=1081.635,112.423,432.792,174.459,22.019,153.712
C05138=1081.629,112.174,432.811,174.457,22.016,153.712
C05139=1081.624,111.924,432.830,174.456,22.014,153.712
C05140=1081.618,111.645,432.851,174.454,22.012,153.712
C05141=1081.612,111.364,432.872,174.451,22.010,153.712
C05142=1081.605,111.085,432.894,174.449,22.007,153.712
C05143=1081.599,110.805,432.915,174.447,22.004,153.711
C05144=1081.593,110.555,432.934,174.446,22.002,153.711
C05145=1081.587,110.307,432.952,174.443,22.000,153.711
C05146=1081.581,110.057,432.971,174.442,21.998,153.711
C05147=1081.576,109.808,432.991,174.440,21.996,153.711
C05148=1081.570,109.559,433.009,174.438,21.994,153.711
C05149=1081.564,109.309,433.027,174.436,21.992,153.710
C05150=1081.559,109.060,433.047,174.435,21.990,153.710
C05151=1081.552,108.811,433.065,174.432,21.987,153.710
C05152=1081.547,108.562,433.084,174.431,21.985,153.710
C05153=1081.541,108.313,433.103,174.429,21.983,153.710
C05154=1081.535,108.063,433.121,174.427,21.981,153.710
C05155=1081.530,107.814,433.140,174.425,21.979,153.710
C05156=1081.524,107.565,433.159,174.424,21.977,153.709
C05157=1081.519,107.316,433.178,174.421,21.975,153.709
C05158=1081.513,107.066,433.196,174.420,21.973,153.709
C05159=1081.507,106.817,433.215,174.418,21.970,153.709
C05160=1081.502,106.568,433.234,174.416,21.968,153.709
C05161=1081.496,106.319,433.252,174.414,21.966,153.709
C05162=1081.490,106.069,433.271,174.413,21.964,153.708
C05163=1081.485,105.821,433.290,174.411,21.962,153.708
C05164=1081.479,105.571,433.308,174.409,21.960,153.708
C05165=1081.473,105.321,433.327,174.407,21.958,153.708
C05166=1081.467,105.073,433.345,174.406,21.956,153.708
C05167=1081.462,104.823,433.364,174.403,21.953,153.708
C05168=1081.457,104.574,433.383,174.402,21.951,153.707
C05169=1081.451,104.325,433.401,174.400,21.948,153.707
C05170=1081.446,104.076,433.420,174.399,21.947,153.707
C05171=1081.439,103.827,433.438,174.396,21.944,153.707
C05172=1081.434,103.576,433.457,174.395,21.942,153.707
C05173=1081.428,103.328,433.475,174.393,21.940,153.707
C05174=1081.422,103.079,433.494,174.391,21.938,153.706
C05175=1081.418,102.829,433.512,174.389,21.936,153.706
C05176=1081.411,102.580,433.531,174.388,21.934,153.706
C05177=1081.406,102.331,433.549,174.385,21.931,153.706
C05178=1081.400,102.082,433.568,174.384,21.929,153.706
C05179=1081.395,101.832,433.586,174.382,21.927,153.706
C05180=1081.389,101.583,433.605,174.381,21.925,153.705
C05181=1081.383,101.333,433.623,174.378,21.922,153.705
C05182=1081.378,101.085,433.642,174.377,21.920,153.705
C05183=1081.372,100.835,433.660,174.375,21.918,153.705
C05184=1081.366,100.586,433.678,174.373,21.916,153.705
C05185=1081.360,100.337,433.696,174.371,21.914,153.705
C05186=1081.355,100.088,433.715,174.370,21.912,153.704
C05187=1081.349,99.838,433.733,174.367,21.910,153.704
C05188=1081.343,99.589,433.752,174.366,21.907,153.704
C05189=1081.338,99.340,433.770,174.364,21.905,153.704
C05190=1081.331,99.090,433.789,174.363,21.903,153.704
C05191=1081.327,98.841,433.807,174.360,21.901,153.704
C05192=1081.320,98.592,433.825,174.359,21.899,153.703
C05193=1081.315,98.343,433.843,174.357,21.896,153.703
C05194=1081.309,98.093,433.861,174.355,21.894,153.703
C05195=1081.303,97.845,433.880,174.353,21.892,153.703
C05196=1081.297,97.595,433.898,174.352,21.890,153.703
C05197=1081.292,97.346,433.917,174.350,21.887,153.703
C05198=1081.286,97.096,433.935,174.348,21.885,153.702
C05199=1081.281,96.847,433.952,174.347,21.883,153.702
C05200=1081.275,96.598,433.971,174.345,21.881,153.702
C05201=1081.269,96.349,433.989,174.343,21.879,153.702
C05202=1081.263,96.099,434.007,174.341,21.877,153.702
C05203=1081.258,95.850,434.026,174.340,21.875,153.702
C05204=1081.251,95.570,434.046,174.338,21.872,153.701
C05205=1081.245,95.291,434.066,174.335,21.870,153.701
C05206=1081.238,95.011,434.087,174.333,21.867,153.701
C05207=1081.233,94.730,434.107,174.332,21.865,153.701
C05208=1081.226,94.481,434.125,174.330,21.862,153.701
C05209=1081.221,94.232,434.143,174.329,21.860,153.700
C05210=1081.215,93.983,434.160,174.326,21.858,153.700
C05211=1081.210,93.734,434.180,174.325,21.856,153.700
C05212=1081.204,93.485,434.197,174.323,21.853,153.700
C05213=1081.198,93.235,434.215,174.321,21.851,153.700
C05214=1081.193,92.986,434.233,174.319,21.849,153.699
C05215=1081.187,92.736,434.251,174.318,21.847,153.699
C05216=1081.181,92.487,434.270,174.317,21.845,153.699
C05217=1081.176,92.238,434.287,174.314,21.842,153.699
C05218=1081.170,91.988,434.306,174.313,21.840,153.699
C05219=1081.165,91.739,434.323,174.311,21.838,153.698
C05220=1081.159,91.490,434.341,174.309,21.836,153.698
C05221=1081.153,91.241,434.359,174.307,21.833,153.698
C05222=1081.148,90.992,434.378,174.306,21.831,153.698
C05223=1081.142,90.742,434.396,174.304,21.828,153.698
C05224=1081.137,90.493,434.413,174.302,21.827,153.698
C05225=1081.130,90.243,434.431,174.300,21.824,153.697
C05226=1081.125,89.994,434.449,174.299,21.822,153.697
C05227=1081.119,89.745,434.467,174.297,21.820,153.697
C05228=1081.113,89.495,434.484,174.295,21.818,153.697
C05229=1081.107,89.246,434.503,174.294,21.816,153.697
C05230=1081.101,88.997,434.520,174.292,21.813,153.696
C05231=1081.096,88.748,434.538,174.290,21.811,153.696
C05232=1081.090,88.499,434.556,174.288,21.809,153.696
C05233=1081.084,88.249,434.573,174.287,21.807,153.696
C05234=1081.078,88.000,434.591,174.285,21.805,153.696
C05235=1081.073,87.751,434.609,174.283,21.802,153.696
C05236=1081.067,87.502,434.626,174.282,21.800,153.695
C05237=1081.061,87.252,434.644,174.280,21.798,153.695
C05238=1081.055,87.003,434.662,174.278,21.796,153.695
C05239=1081.049,86.753,434.680,174.276,21.794,153.695
C05240=1081.044,86.504,434.698,174.275,21.791,153.695
C05241=1081.039,86.255,434.716,174.274,21.789,153.694
C05242=1081.033,86.005,434.734,174.271,21.787,153.694
C05243=1081.027,85.756,434.751,174.270,21.785,153.694
C05244=1081.022,85.507,434.769,174.268,21.782,153.694
C05245=1081.016,85.257,434.787,174.267,21.780,153.694
C05246=1081.010,85.008,434.804,174.264,21.778,153.694
C05247=1081.005,84.759,434.822,174.263,21.776,153.693
C05248=1080.999,84.509,434.840,174.262,21.773,153.693
C05249=1080.993,84.260,434.857,174.260,21.771,153.693
C05250=1080.987,84.011,434.875,174.258,21.769,153.693
C05251=1080.981,83.762,434.893,174.256,21.767,153.693
C05252=1080.976,83.512,434.910,174.255,21.764,153.692
C05253=1080.971,83.263,434.927,174.253,21.762,153.692
C05254=1080.964,83.013,434.944,174.251,21.760,153.692
C05255=1080.958,82.764,434.962,174.250,21.758,153.692
C05256=1080.953,82.515,434.980,174.248,21.755,153.692
C05257=1080.947,82.266,434.997,174.246,21.753,153.691
C05258=1080.941,82.017,435.015,174.244,21.751,153.691
C05259=1080.936,81.767,435.032,174.243,21.748,153.691
C05260=1080.930,81.518,435.050,174.242,21.747,153.691
C05261=1080.924,81.268,435.067,174.239,21.744,153.691
C05262=1080.919,81.019,435.085,174.238,21.742,153.690
C05263=1080.913,80.770,435.103,174.236,21.739,153.690
C05264=1080.908,80.521,435.120,174.235,21.737,153.690
C05265=1080.902,80.271,435.137,174.233,21.735,153.690
C05266=1080.896,80.022,435.155,174.231,21.733,153.690
C05267=1080.891,79.773,435.173,174.230,21.731,153.689
C05268=1080.884,79.493,435.192,174.228,21.728,153.689
C05269=1080.878,79.213,435.211,174.226,21.725,153.689
C05270=1080.872,78.933,435.231,174.224,21.723,153.689
C05271=1080.866,78.653,435.250,174.222,21.720,153.689
C05272=1080.860,78.404,435.268,174.220,21.718,153.688
C05273=1080.854,78.155,435.286,174.219,21.716,153.688
C05274=1080.848,77.906,435.303,174.218,21.713,153.688
C05275=1080.843,77.656,435.319,174.215,21.711,153.688
C05276=1080.837,77.407,435.337,174.214,21.709,153.688
C05277=1080.831,77.157,435.355,174.212,21.706,153.687
C05278=1080.825,76.908,435.371,174.211,21.704,153.687
C05279=1080.820,76.659,435.389,174.209,21.702,153.687
C05280=1080.813,76.409,435.407,174.207,21.699,153.687
C05281=1080.808,76.160,435.424,174.206,21.698,153.687
C05282=1080.802,75.911,435.441,174.204,21.695,153.686
C05283=1080.796,75.662,435.458,174.202,21.693,153.686
C05284=1080.791,75.412,435.475,174.201,21.691,153.686
C05285=1080.785,75.163,435.493,174.199,21.688,153.686
C05286=1080.779,74.913,435.509,174.197,21.686,153.686
C05287=1080.774,74.664,435.527,174.196,21.684,153.685
C05288=1080.768,74.415,435.544,174.194,21.682,153.685
C05289=1080.762,74.165,435.561,174.193,21.680,153.685
C05290=1080.756,73.916,435.578,174.191,21.677,153.685
C05291=1080.751,73.666,435.595,174.189,21.675,153.685
C05292=1080.745,73.417,435.613,174.188,21.672,153.684
C05293=1080.739,73.168,435.629,174.186,21.670,153.684
C05294=1080.733,72.918,435.647,174.185,21.668,153.684
C05295=1080.728,72.669,435.665,174.182,21.665,153.684
C05296=1080.722,72.420,435.681,174.181,21.663,153.684
C05297=1080.716,72.171,435.698,174.180,21.661,153.683
C05298=1080.711,71.921,435.715,174.178,21.659,153.683
C05299=1080.705,71.672,435.732,174.176,21.657,153.683
C05300=1080.699,71.422,435.750,174.175,21.655,153.683
C05301=1080.693,71.173,435.767,174.173,21.652,153.683
C05302=1080.688,70.924,435.783,174.172,21.650,153.682
C05303=1080.682,70.675,435.801,174.170,21.647,153.682
C05304=1080.677,70.425,435.818,174.168,21.645,153.682
C05305=1080.671,70.176,435.834,174.167,21.643,153.682
C05306=1080.665,69.927,435.852,174.165,21.640,153.681
C05307=1080.659,69.677,435.868,174.163,21.638,153.681
C05308=1080.653,69.427,435.886,174.161,21.636,153.681
C05309=1080.647,69.178,435.902,174.160,21.633,153.681
C05310=1080.642,68.929,435.920,174.159,21.631,153.681
C05311=1080.637,68.679,435.936,174.156,21.629,153.681
C05312=1080.631,68.430,435.953,174.155,21.627,153.680
C05313=1080.625,68.181,435.970,174.154,21.625,153.680
C05314=1080.619,67.932,435.987,174.152,21.622,153.680
C05315=1080.614,67.682,436.003,174.151,21.620,153.680
C05316=1080.607,67.433,436.021,174.149,21.618,153.679
C05317=1080.602,67.183,436.038,174.147,21.615,153.679
C05318=1080.596,66.934,436.055,174.146,21.613,153.679
C05319=1080.590,66.685,436.071,174.144,21.611,153.679
C05320=1080.584,66.435,436.088,174.142,21.608,153.679
C05321=1080.579,66.186,436.104,174.141,21.606,153.678
C05322=1080.573,65.937,436.121,174.139,21.603,153.678
C05323=1080.568,65.687,436.138,174.138,21.602,153.678
C05324=1080.562,65.438,436.155,174.136,21.600,153.678
C05325=1080.556,65.189,436.172,174.134,21.597,153.678
C05326=1080.550,64.939,436.189,174.133,21.595,153.677
C05327=1080.544,64.689,436.205,174.132,21.592,153.677
C05328=1080.539,64.440,436.222,174.130,21.590,153.677
C05329=1080.532,64.191,436.239,174.128,21.588,153.677
C05330=1080.527,63.941,436.256,174.126,21.585,153.677
C05331=1080.521,63.692,436.272,174.125,21.583,153.676
C05332=1080.514,63.412,436.290,174.123,21.580,153.676
C05333=1080.508,63.133,436.309,174.121,21.578,153.676
C05334=1080.501,62.853,436.329,174.119,21.575,153.676
C05335=1080.495,62.573,436.346,174.118,21.573,153.675
C05336=1080.489,62.323,436.363,174.116,21.571,153.675
C05337=1080.483,62.074,436.380,174.115,21.569,153.675
C05338=1080.477,61.825,436.396,174.112,21.566,153.675
C05339=1080.471,61.575,436.413,174.111,21.564,153.675
C05340=1080.465,61.326,436.429,174.110,21.562,153.674
C05341=1080.460,61.076,436.446,174.108,21.559,153.674
C05342=1080.453,60.826,436.462,174.107,21.557,153.674
C05343=1080.447,60.578,436.479,174.105,21.555,153.674
C05344=1080.441,60.328,436.496,174.103,21.552,153.674
C05345=1080.436,60.079,436.512,174.102,21.550,153.673
C05346=1080.430,59.829,436.529,174.100,21.548,153.673
C05347=1080.424,59.580,436.545,174.098,21.545,153.673
C05348=1080.418,59.331,436.561,174.097,21.543,153.673
C05349=1080.413,59.081,436.578,174.096,21.542,153.673
C05350=1080.407,58.832,436.594,174.094,21.539,153.672
C05351=1080.401,58.582,436.611,174.092,21.537,153.672
C05352=1080.395,58.333,436.627,174.091,21.534,153.672
C05353=1080.389,58.084,436.643,174.089,21.532,153.672
C05354=1080.384,57.835,436.661,174.088,21.530,153.672
C05355=1080.378,57.585,436.677,174.086,21.527,153.671
C05356=1080.372,57.336,436.693,174.084,21.525,153.671
C05357=1080.366,57.086,436.709,174.083,21.523,153.671
C05358=1080.360,56.837,436.726,174.082,21.521,153.671
C05359=1080.355,56.587,436.743,174.080,21.518,153.671
C05360=1080.349,56.338,436.759,174.078,21.516,153.670
C05361=1080.343,56.089,436.775,174.077,21.514,153.670
C05362=1080.337,55.839,436.791,174.075,21.511,153.670
C05363=1080.331,55.590,436.808,174.074,21.509,153.670
C05364=1080.326,55.340,436.824,174.072,21.507,153.669
C05365=1080.320,55.090,436.840,174.070,21.504,153.669
C05366=1080.314,54.841,436.856,174.069,21.502,153.669
C05367=1080.308,54.592,436.872,174.068,21.500,153.669
C05368=1080.302,54.342,436.889,174.066,21.497,153.669
C05369=1080.297,54.094,436.905,174.064,21.495,153.668
C05370=1080.292,53.844,436.921,174.063,21.493,153.668
C05371=1080.286,53.595,436.938,174.061,21.490,153.668
C05372=1080.280,53.345,436.954,174.060,21.488,153.668
C05373=1080.274,53.096,436.970,174.059,21.486,153.667
C05374=1080.268,52.847,436.987,174.056,21.483,153.667
C05375=1080.262,52.597,437.003,174.055,21.481,153.667
C05376=1080.257,52.347,437.019,174.054,21.479,153.667
C05377=1080.251,52.098,437.035,174.052,21.477,153.667
C05378=1080.245,51.848,437.051,174.050,21.474,153.666
C05379=1080.239,51.599,437.068,174.049,21.472,153.666
C05380=1080.234,51.350,437.084,174.047,21.469,153.666
C05381=1080.228,51.101,437.100,174.046,21.467,153.666
C05382=1080.222,50.851,437.115,174.045,21.465,153.665
C05383=1080.216,50.602,437.132,174.042,21.462,153.665
C05384=1080.211,50.352,437.148,174.041,21.460,153.665
C05385=1080.205,50.103,437.165,174.040,21.458,153.665
C05386=1080.199,49.853,437.181,174.038,21.455,153.665
C05387=1080.194,49.604,437.196,174.036,21.453,153.664
C05388=1080.188,49.355,437.212,174.035,21.451,153.664
C05389=1080.182,49.105,437.229,174.033,21.448,153.664
C05390=1080.176,48.856,437.245,174.032,21.446,153.664
C05391=1080.170,48.606,437.260,174.031,21.444,153.663
C05392=1080.164,48.357,437.277,174.029,21.441,153.663
C05393=1080.159,48.108,437.293,174.027,21.438,153.663
C05394=1080.154,47.858,437.309,174.026,21.437,153.663
C05395=1080.148,47.608,437.325,174.025,21.434,153.662
C05396=1080.141,47.328,437.343,174.023,21.432,153.662
C05397=1080.135,47.048,437.361,174.021,21.429,153.662
C05398=1080.129,46.768,437.379,174.020,21.426,153.662
C05399=1080.122,46.489,437.397,174.018,21.423,153.661
C05400=1080.116,46.239,437.413,174.016,21.421,153.661
C05401=1080.111,45.989,437.429,174.015,21.419,153.661
C05402=1080.105,45.740,437.444,174.013,21.416,153.661
C05403=1080.100,45.491,437.461,174.012,21.414,153.661
C05404=1080.094,45.241,437.477,174.011,21.412,153.660
C05405=1080.089,44.991,437.493,174.008,21.409,153.660
C05406=1080.083,44.743,437.509,174.007,21.407,153.660
C05407=1080.077,44.493,437.525,174.006,21.404,153.660
C05408=1080.072,44.243,437.540,174.004,21.402,153.659
C05409=1080.066,43.994,437.557,174.003,21.399,153.659
C05410=1080.061,43.745,437.572,174.001,21.397,153.659
C05411=1080.055,43.495,437.588,174.000,21.395,153.659
C05412=1080.049,43.246,437.604,173.998,21.393,153.658
C05413=1080.042,42.996,437.619,173.997,21.390,153.658
C05414=1080.036,42.747,437.635,173.996,21.388,153.658
C05415=1080.031,42.498,437.651,173.993,21.385,153.658
C05416=1080.025,42.248,437.667,173.992,21.383,153.658
C05417=1080.020,41.998,437.682,173.991,21.381,153.657
C05418=1080.014,41.749,437.699,173.989,21.378,153.657
C05419=1080.008,41.499,437.714,173.988,21.376,153.657
C05420=1080.002,41.251,437.730,173.986,21.374,153.657
C05421=1079.997,41.001,437.745,173.985,21.372,153.656
C05422=1079.991,40.751,437.761,173.983,21.369,153.656
C05423=1079.985,40.501,437.777,173.982,21.367,153.656
C05424=1079.980,40.253,437.793,173.980,21.365,153.656
C05425=1079.974,40.003,437.808,173.978,21.362,153.656
C05426=1079.967,39.754,437.824,173.977,21.360,153.655
C05427=1079.962,39.505,437.839,173.976,21.357,153.655
C05428=1079.956,39.255,437.855,173.974,21.355,153.655
C05429=1079.951,39.005,437.871,173.973,21.353,153.655
C05430=1079.945,38.755,437.886,173.971,21.351,153.654
C05431=1079.940,38.507,437.902,173.970,21.348,153.654
C05432=1079.933,38.257,437.917,173.968,21.346,153.654
C05433=1079.927,38.008,437.934,173.967,21.343,153.654
C05434=1079.922,37.758,437.949,173.965,21.341,153.654
C05435=1079.917,37.508,437.964,173.963,21.338,153.653
C05436=1079.910,37.259,437.980,173.962,21.336,153.653
C05437=1079.904,37.009,437.995,173.961,21.334,153.653
C05438=1079.899,36.761,438.011,173.960,21.332,153.653
C05439=1079.893,36.511,438.026,173.958,21.329,153.652
C05440=1079.887,36.261,438.042,173.956,21.327,153.652
C05441=1079.880,36.012,438.058,173.955,21.325,153.652
C05442=1079.875,35.763,438.073,173.953,21.322,153.652
C05443=1079.869,35.513,438.088,173.952,21.320,153.651
C05444=1079.863,35.264,438.104,173.950,21.318,153.651
C05445=1079.858,35.014,438.119,173.949,21.315,153.651
C05446=1079.852,34.765,438.135,173.947,21.313,153.651
C05447=1079.846,34.515,438.150,173.946,21.311,153.651
C05448=1079.840,34.266,438.166,173.945,21.309,153.650
C05449=1079.835,34.016,438.181,173.943,21.306,153.650
C05450=1079.828,33.767,438.196,173.941,21.304,153.650
C05451=1079.822,33.517,438.212,173.940,21.302,153.650
C05452=1079.817,33.268,438.227,173.939,21.299,153.649
C05453=1079.811,33.018,438.242,173.937,21.297,153.649
C05454=1079.805,32.768,438.258,173.935,21.294,153.649
C05455=1079.799,32.520,438.273,173.934,21.292,153.649
C05456=1079.794,32.270,438.289,173.933,21.290,153.649
C05457=1079.788,32.021,438.303,173.931,21.287,153.648
C05458=1079.782,31.771,438.319,173.930,21.285,153.648
C05459=1079.777,31.521,438.334,173.929,21.283,153.648
C05460=1079.770,31.242,438.351,173.926,21.280,153.648
C05461=1079.763,30.961,438.368,173.925,21.278,153.647
C05462=1079.757,30.682,438.386,173.923,21.275,153.647
